gfCNCPoint6[4861] = {X 129.4526, Y 19.2665, Z -8.0000, A 0.000, B 0.000, C 0.000 }
gfCNCPoint6[4862] = {X 129.1449, Y 18.3872, Z -8.0000, A 0.000, B 0.000, C 0.000 }
gfCNCPoint6[4863] = {X 129.0406, Y 17.4615, Z -8.0000, A 0.000, B 0.000, C 0.000 }
gfCNCPoint6[4864] = {X 129.0406, Y 10.4835, Z -8.0000, A 0.000, B 0.000, C 0.000 }
gfCNCPoint6[4865] = {X 129.1435, Y 9.5642, Z -8.0000, A 0.000, B 0.000, C 0.000 }
gfCNCPoint6[4866] = {X 129.4469, Y 8.6904, Z -8.0000, A 0.000, B 0.000, C 0.000 }
gfCNCPoint6[4867] = {X 129.9360, Y 7.9052, Z -8.0000, A 0.000, B 0.000, C 0.000 }
gfCNCPoint6[4868] = {X 130.5864, Y 7.2475, Z -8.0000, A 0.000, B 0.000, C 0.000 }
gfCNCPoint6[4869] = {X 131.3662, Y 6.7499, Z -8.0000, A 0.000, B 0.000, C 0.000 }
gfCNCPoint6[4870] = {X 132.2366, Y 6.4368, Z -8.0000, A 0.000, B 0.000, C 0.000 }
gfCNCPoint6[4871] = {X 133.1547, Y 6.3238, Z -8.0000, A 0.000, B 0.000, C 0.000 }
gfCNCPoint6[4872] = {X 133.8850, Y 6.3237, Z -8.0000, A 0.000, B 0.000, C 0.000 }
gfCNCPoint6[4873] = {X 134.6950, Y 6.4118, Z -8.0000, A 0.000, B 0.000, C 0.000 }
gfCNCPoint6[4874] = {X 135.4723, Y 6.6562, Z -8.0000, A 0.000, B 0.000, C 0.000 }
gfCNCPoint6[4875] = {X 136.1871, Y 7.0473, Z -8.0000, A 0.000, B 0.000, C 0.000 }
gfCNCPoint6[4876] = {X 136.8119, Y 7.5703, Z -8.0000, A 0.000, B 0.000, C 0.000 }
gfCNCPoint6[4877] = {X 137.3228, Y 8.2050, Z -8.0000, A 0.000, B 0.000, C 0.000 }
gfCNCPoint6[4878] = {X 155.1990, Y 8.2064, Z -8.0000, A 0.000, B 0.000, C 0.000 }
gfCNCPoint6[4879] = {X 155.7105, Y 7.5705, Z -8.0000, A 0.000, B 0.000, C 0.000 }
gfCNCPoint6[4880] = {X 156.3364, Y 7.0468, Z -8.0000, A 0.000, B 0.000, C 0.000 }
gfCNCPoint6[4881] = {X 157.0525, Y 6.6553, Z -8.0000, A 0.000, B 0.000, C 0.000 }
gfCNCPoint6[4882] = {X 157.8313, Y 6.4111, Z -8.0000, A 0.000, B 0.000, C 0.000 }
gfCNCPoint6[4883] = {X 158.6427, Y 6.3237, Z -8.0000, A 0.000, B 0.000, C 0.000 }
gfCNCPoint6[4884] = {X 159.3760, Y 6.3239, Z -8.0000, A 0.000, B 0.000, C 0.000 }
gfCNCPoint6[4885] = {X 160.2928, Y 6.4383, Z -8.0000, A 0.000, B 0.000, C 0.000 }
gfCNCPoint6[4886] = {X 161.1617, Y 6.7524, Z -8.0000, A 0.000, B 0.000, C 0.000 }
gfCNCPoint6[4887] = {X 161.9398, Y 7.2504, Z -8.0000, A 0.000, B 0.000, C 0.000 }
gfCNCPoint6[4888] = {X 162.5889, Y 7.9079, Z -8.0000, A 0.000, B 0.000, C 0.000 }
gfCNCPoint6[4889] = {X 163.0768, Y 8.6925, Z -8.0000, A 0.000, B 0.000, C 0.000 }
gfCNCPoint6[4890] = {X 163.3795, Y 9.5653, Z -8.0000, A 0.000, B 0.000, C 0.000 }
gfCNCPoint6[4891] = {X 163.4821, Y 10.4835, Z -8.0000, A 0.000, B 0.000, C 0.000 }
gfCNCPoint6[4892] = {X 163.4821, Y 17.4615, Z -8.0000, A 0.000, B 0.000, C 0.000 }
gfCNCPoint6[4893] = {X 163.3795, Y 18.3798, Z -8.0000, A 0.000, B 0.000, C 0.000 }
gfCNCPoint6[4894] = {X 163.0767, Y 19.2527, Z -8.0000, A 0.000, B 0.000, C 0.000 }
gfCNCPoint6[4895] = {X 162.5887, Y 20.0373, Z -8.0000, A 0.000, B 0.000, C 0.000 }
gfCNCPoint6[4896] = {X 161.9396, Y 20.6948, Z -8.0000, A 0.000, B 0.000, C 0.000 }
gfCNCPoint6[4897] = {X 161.1613, Y 21.1929, Z -8.0000, A 0.000, B 0.000, C 0.000 }
gfCNCPoint6[4898] = {X 160.2923, Y 21.5068, Z -8.0000, A 0.000, B 0.000, C 0.000 }
gfCNCPoint6[4899] = {X 159.3755, Y 21.6212, Z -8.0000, A 0.000, B 0.000, C 0.000 }
gfCNCPoint6[4900] = {X 158.6800, Y 21.6215, Z -8.0000, A 0.000, B 0.000, C 0.000 }
gfCNCPoint6[4901] = {X 157.8559, Y 21.5370, Z -8.0000, A 0.000, B 0.000, C 0.000 }
gfCNCPoint6[4902] = {X 157.0645, Y 21.2919, Z -8.0000, A 0.000, B 0.000, C 0.000 }
gfCNCPoint6[4903] = {X 156.3369, Y 20.8959, Z -8.0000, A 0.000, B 0.000, C 0.000 }
gfCNCPoint6[4904] = {X 155.7014, Y 20.3644, Z -8.0000, A 0.000, B 0.000, C 0.000 }
gfCNCPoint6[4905] = {X 155.1830, Y 19.7182, Z -8.0000, A 0.000, B 0.000, C 0.000 }
gfCNCPoint6[4906] = {X 152.1174, Y 19.7191, Z -8.0000, A 0.000, B 0.000, C 0.000 }
gfCNCPoint6[4907] = {X 152.1164, Y 40.9370, Z -8.0000, A 0.000, B 0.000, C 0.000 }
gfCNCPoint6[4908] = {X 152.6208, Y 41.4801, Z -8.0000, A 0.000, B 0.000, C 0.000 }
gfCNCPoint6[4909] = {X 152.7136, Y 41.5904, Z -8.0000, A 0.000, B 0.000, C 0.000 }
gfCNCPoint6[4910] = {X 153.2194, Y 42.3850, Z -8.0000, A 0.000, B 0.000, C 0.000 }
gfCNCPoint6[4911] = {X 153.5346, Y 43.2727, Z -8.0000, A 0.000, B 0.000, C 0.000 }
gfCNCPoint6[4912] = {X 153.6431, Y 44.2084, Z -8.0000, A 0.000, B 0.000, C 0.000 }
gfCNCPoint6[4913] = {X 153.6429, Y 45.0400, Z -8.0000, A 0.000, B 0.000, C 0.000 }
gfCNCPoint6[4914] = {X 153.5310, Y 45.9591, Z -8.0000, A 0.000, B 0.000, C 0.000 }
gfCNCPoint6[4915] = {X 153.2186, Y 46.8306, Z -8.0000, A 0.000, B 0.000, C 0.000 }
gfCNCPoint6[4916] = {X 152.7212, Y 47.6115, Z -8.0000, A 0.000, B 0.000, C 0.000 }
gfCNCPoint6[4917] = {X 152.0634, Y 48.2631, Z -8.0000, A 0.000, B 0.000, C 0.000 }
gfCNCPoint6[4918] = {X 151.2778, Y 48.7530, Z -8.0000, A 0.000, B 0.000, C 0.000 }
gfCNCPoint6[4919] = {X 150.4032, Y 49.0570, Z -8.0000, A 0.000, B 0.000, C 0.000 }
gfCNCPoint6[4920] = {X 149.4831, Y 49.1600, Z -8.0000, A 0.000, B 0.000, C 0.000 }
gfCNCPoint6[4921] = {X 143.0396, Y 49.1600, Z -8.0000, A 0.000, B 0.000, C 0.000 }
gfCNCPoint6[4922] = {X 142.1185, Y 49.0567, Z -8.0000, A 0.000, B 0.000, C 0.000 }
gfCNCPoint6[4923] = {X 141.2432, Y 48.7521, Z -8.0000, A 0.000, B 0.000, C 0.000 }
gfCNCPoint6[4924] = {X 140.4570, Y 48.2612, Z -8.0000, A 0.000, B 0.000, C 0.000 }
gfCNCPoint6[4925] = {X 139.7990, Y 47.6084, Z -8.0000, A 0.000, B 0.000, C 0.000 }
gfCNCPoint6[4926] = {X 139.3019, Y 46.8261, Z -8.0000, A 0.000, B 0.000, C 0.000 }
gfCNCPoint6[4927] = {X 138.9903, Y 45.9532, Z -8.0000, A 0.000, B 0.000, C 0.000 }
gfCNCPoint6[4928] = {X 138.8798, Y 45.0329, Z -8.0000, A 0.000, B 0.000, C 0.000 }
gfCNCPoint6[4929] = {X 138.8800, Y 44.1516, Z -8.0000, A 0.000, B 0.000, C 0.000 }
gfCNCPoint6[4930] = {X 138.9906, Y 43.2545, Z -8.0000, A 0.000, B 0.000, C 0.000 }
gfCNCPoint6[4931] = {X 139.2922, Y 42.4026, Z -8.0000, A 0.000, B 0.000, C 0.000 }
gfCNCPoint6[4932] = {X 139.7708, Y 41.6358, Z -8.0000, A 0.000, B 0.000, C 0.000 }
gfCNCPoint6[4933] = {X 140.4036, Y 40.9906, Z -8.0000, A 0.000, B 0.000, C 0.000 }
gfCNCPoint6[4934] = {X 140.4036, Y 30.3971, Z -8.0000, A 0.000, B 0.000, C 0.000 }
gfCNCPoint6[4935] = {X 136.4036, Y 30.3971, Z -8.0000, A 0.000, B 0.000, C 0.000 }
gfCNCPoint6[4936] = {X 140.4836, Y 30.3971, Z -8.0000, A 0.000, B 0.000, C 0.000 }
gfCNCPoint6[4937] = {X 140.4836, Y 19.6385, Z -8.0000, A 0.000, B 0.000, C 0.000 }
gfCNCPoint6[4938] = {X 137.2911, Y 19.6382, Z -8.0000, A 0.000, B 0.000, C 0.000 }
gfCNCPoint6[4939] = {X 137.2218, Y 19.7475, Z -8.0000, A 0.000, B 0.000, C 0.000 }
gfCNCPoint6[4940] = {X 136.5756, Y 20.4907, Z -8.0000, A 0.000, B 0.000, C 0.000 }
gfCNCPoint6[4941] = {X 135.7702, Y 21.0573, Z -8.0000, A 0.000, B 0.000, C 0.000 }
gfCNCPoint6[4942] = {X 134.8524, Y 21.4145, Z -8.0000, A 0.000, B 0.000, C 0.000 }
gfCNCPoint6[4943] = {X 133.8758, Y 21.5414, Z -8.0000, A 0.000, B 0.000, C 0.000 }
gfCNCPoint6[4944] = {X 133.2006, Y 21.5415, Z -8.0000, A 0.000, B 0.000, C 0.000 }
gfCNCPoint6[4945] = {X 132.2928, Y 21.4392, Z -8.0000, A 0.000, B 0.000, C 0.000 }
gfCNCPoint6[4946] = {X 131.4304, Y 21.1375, Z -8.0000, A 0.000, B 0.000, C 0.000 }
gfCNCPoint6[4947] = {X 130.6568, Y 20.6514, Z -8.0000, A 0.000, B 0.000, C 0.000 }
gfCNCPoint6[4948] = {X 130.0108, Y 20.0054, Z -8.0000, A 0.000, B 0.000, C 0.000 }
gfCNCPoint6[4949] = {X 129.5247, Y 19.2318, Z -8.0000, A 0.000, B 0.000, C 0.000 }
gfCNCPoint6[4950] = {X 129.2229, Y 18.3694, Z -8.0000, A 0.000, B 0.000, C 0.000 }
gfCNCPoint6[4951] = {X 129.1206, Y 17.4615, Z -8.0000, A 0.000, B 0.000, C 0.000 }
gfCNCPoint6[4952] = {X 129.1206, Y 10.4835, Z -8.0000, A 0.000, B 0.000, C 0.000 }
gfCNCPoint6[4953] = {X 129.2215, Y 9.5820, Z -8.0000, A 0.000, B 0.000, C 0.000 }
gfCNCPoint6[4954] = {X 129.5191, Y 8.7250, Z -8.0000, A 0.000, B 0.000, C 0.000 }
gfCNCPoint6[4955] = {X 129.9986, Y 7.9550, Z -8.0000, A 0.000, B 0.000, C 0.000 }
gfCNCPoint6[4956] = {X 130.6365, Y 7.3099, Z -8.0000, A 0.000, B 0.000, C 0.000 }
gfCNCPoint6[4957] = {X 131.4011, Y 6.8218, Z -8.0000, A 0.000, B 0.000, C 0.000 }
gfCNCPoint6[4958] = {X 132.2547, Y 6.5147, Z -8.0000, A 0.000, B 0.000, C 0.000 }
gfCNCPoint6[4959] = {X 133.1551, Y 6.4038, Z -8.0000, A 0.000, B 0.000, C 0.000 }
gfCNCPoint6[4960] = {X 133.8841, Y 6.4037, Z -8.0000, A 0.000, B 0.000, C 0.000 }
gfCNCPoint6[4961] = {X 134.6870, Y 6.4919, Z -8.0000, A 0.000, B 0.000, C 0.000 }
gfCNCPoint6[4962] = {X 135.4568, Y 6.7365, Z -8.0000, A 0.000, B 0.000, C 0.000 }
gfCNCPoint6[4963] = {X 136.1633, Y 7.1280, Z -8.0000, A 0.000, B 0.000, C 0.000 }
gfCNCPoint6[4964] = {X 136.7789, Y 7.6510, Z -8.0000, A 0.000, B 0.000, C 0.000 }
gfCNCPoint6[4965] = {X 137.2793, Y 8.2850, Z -8.0000, A 0.000, B 0.000, C 0.000 }
gfCNCPoint6[4966] = {X 155.2425, Y 8.2864, Z -8.0000, A 0.000, B 0.000, C 0.000 }
gfCNCPoint6[4967] = {X 155.2880, Y 8.2168, Z -8.0000, A 0.000, B 0.000, C 0.000 }
gfCNCPoint6[4968] = {X 155.3349, Y 8.1482, Z -8.0000, A 0.000, B 0.000, C 0.000 }
gfCNCPoint6[4969] = {X 155.9800, Y 7.4251, Z -8.0000, A 0.000, B 0.000, C 0.000 }
gfCNCPoint6[4970] = {X 156.7775, Y 6.8745, Z -8.0000, A 0.000, B 0.000, C 0.000 }
gfCNCPoint6[4971] = {X 157.6823, Y 6.5275, Z -8.0000, A 0.000, B 0.000, C 0.000 }
gfCNCPoint6[4972] = {X 158.6434, Y 6.4037, Z -8.0000, A 0.000, B 0.000, C 0.000 }
gfCNCPoint6[4973] = {X 159.3750, Y 6.4039, Z -8.0000, A 0.000, B 0.000, C 0.000 }
gfCNCPoint6[4974] = {X 160.2741, Y 6.5161, Z -8.0000, A 0.000, B 0.000, C 0.000 }
gfCNCPoint6[4975] = {X 161.1263, Y 6.8241, Z -8.0000, A 0.000, B 0.000, C 0.000 }
gfCNCPoint6[4976] = {X 161.8895, Y 7.3126, Z -8.0000, A 0.000, B 0.000, C 0.000 }
gfCNCPoint6[4977] = {X 162.5260, Y 7.9574, Z -8.0000, A 0.000, B 0.000, C 0.000 }
gfCNCPoint6[4978] = {X 163.0046, Y 8.7269, Z -8.0000, A 0.000, B 0.000, C 0.000 }
gfCNCPoint6[4979] = {X 163.3015, Y 9.5830, Z -8.0000, A 0.000, B 0.000, C 0.000 }
gfCNCPoint6[4980] = {X 163.4021, Y 10.4835, Z -8.0000, A 0.000, B 0.000, C 0.000 }
gfCNCPoint6[4981] = {X 163.4021, Y 17.4615, Z -8.0000, A 0.000, B 0.000, C 0.000 }
gfCNCPoint6[4982] = {X 163.3015, Y 18.3621, Z -8.0000, A 0.000, B 0.000, C 0.000 }
gfCNCPoint6[4983] = {X 163.0046, Y 19.2182, Z -8.0000, A 0.000, B 0.000, C 0.000 }
gfCNCPoint6[4984] = {X 162.5260, Y 19.9876, Z -8.0000, A 0.000, B 0.000, C 0.000 }
gfCNCPoint6[4985] = {X 161.8895, Y 20.6325, Z -8.0000, A 0.000, B 0.000, C 0.000 }
gfCNCPoint6[4986] = {X 161.1263, Y 21.1209, Z -8.0000, A 0.000, B 0.000, C 0.000 }
gfCNCPoint6[4987] = {X 160.2741, Y 21.4289, Z -8.0000, A 0.000, B 0.000, C 0.000 }
gfCNCPoint6[4988] = {X 159.3750, Y 21.5412, Z -8.0000, A 0.000, B 0.000, C 0.000 }
gfCNCPoint6[4989] = {X 158.6802, Y 21.5415, Z -8.0000, A 0.000, B 0.000, C 0.000 }
gfCNCPoint6[4990] = {X 157.8634, Y 21.4569, Z -8.0000, A 0.000, B 0.000, C 0.000 }
gfCNCPoint6[4991] = {X 157.0797, Y 21.2114, Z -8.0000, A 0.000, B 0.000, C 0.000 }
gfCNCPoint6[4992] = {X 156.3605, Y 20.8151, Z -8.0000, A 0.000, B 0.000, C 0.000 }
gfCNCPoint6[4993] = {X 155.7345, Y 20.2836, Z -8.0000, A 0.000, B 0.000, C 0.000 }
gfCNCPoint6[4994] = {X 155.2267, Y 19.6382, Z -8.0000, A 0.000, B 0.000, C 0.000 }
gfCNCPoint6[4995] = {X 152.0374, Y 19.6392, Z -8.0000, A 0.000, B 0.000, C 0.000 }
gfCNCPoint6[4996] = {X 152.0364, Y 40.9685, Z -8.0000, A 0.000, B 0.000, C 0.000 }
gfCNCPoint6[4997] = {X 152.5609, Y 41.5331, Z -8.0000, A 0.000, B 0.000, C 0.000 }
gfCNCPoint6[4998] = {X 152.6518, Y 41.6413, Z -8.0000, A 0.000, B 0.000, C 0.000 }
gfCNCPoint6[4999] = {X 153.1477, Y 42.4206, Z -8.0000, A 0.000, B 0.000, C 0.000 }
gfCNCPoint6[5000] = {X 153.4567, Y 43.2911, Z -8.0000, A 0.000, B 0.000, C 0.000 }
gfCNCPoint6[5001] = {X 153.5631, Y 44.2086, Z -8.0000, A 0.000, B 0.000, C 0.000 }
gfCNCPoint6[5002] = {X 153.5629, Y 45.0392, Z -8.0000, A 0.000, B 0.000, C 0.000 }
gfCNCPoint6[5003] = {X 153.4532, Y 45.9406, Z -8.0000, A 0.000, B 0.000, C 0.000 }
gfCNCPoint6[5004] = {X 153.1468, Y 46.7954, Z -8.0000, A 0.000, B 0.000, C 0.000 }
gfCNCPoint6[5005] = {X 152.6589, Y 47.5613, Z -8.0000, A 0.000, B 0.000, C 0.000 }
gfCNCPoint6[5006] = {X 152.0138, Y 48.2003, Z -8.0000, A 0.000, B 0.000, C 0.000 }
gfCNCPoint6[5007] = {X 151.2432, Y 48.6808, Z -8.0000, A 0.000, B 0.000, C 0.000 }
gfCNCPoint6[5008] = {X 150.3855, Y 48.9789, Z -8.0000, A 0.000, B 0.000, C 0.000 }
gfCNCPoint6[5009] = {X 149.4831, Y 49.0800, Z -8.0000, A 0.000, B 0.000, C 0.000 }
gfCNCPoint6[5010] = {X 143.0396, Y 49.0800, Z -8.0000, A 0.000, B 0.000, C 0.000 }
gfCNCPoint6[5011] = {X 142.1362, Y 48.9787, Z -8.0000, A 0.000, B 0.000, C 0.000 }
gfCNCPoint6[5012] = {X 141.2777, Y 48.6799, Z -8.0000, A 0.000, B 0.000, C 0.000 }
gfCNCPoint6[5013] = {X 140.5066, Y 48.1985, Z -8.0000, A 0.000, B 0.000, C 0.000 }
gfCNCPoint6[5014] = {X 139.8613, Y 47.5582, Z -8.0000, A 0.000, B 0.000, C 0.000 }
gfCNCPoint6[5015] = {X 139.3737, Y 46.7910, Z -8.0000, A 0.000, B 0.000, C 0.000 }
gfCNCPoint6[5016] = {X 139.0682, Y 45.9349, Z -8.0000, A 0.000, B 0.000, C 0.000 }
gfCNCPoint6[5017] = {X 138.9598, Y 45.0323, Z -8.0000, A 0.000, B 0.000, C 0.000 }
gfCNCPoint6[5018] = {X 138.9600, Y 44.1527, Z -8.0000, A 0.000, B 0.000, C 0.000 }
gfCNCPoint6[5019] = {X 139.0706, Y 43.2637, Z -8.0000, A 0.000, B 0.000, C 0.000 }
gfCNCPoint6[5020] = {X 139.3725, Y 42.4203, Z -8.0000, A 0.000, B 0.000, C 0.000 }
gfCNCPoint6[5021] = {X 139.8512, Y 41.6631, Z -8.0000, A 0.000, B 0.000, C 0.000 }
gfCNCPoint6[5022] = {X 140.4836, Y 41.0287, Z -8.0000, A 0.000, B 0.000, C 0.000 }
gfCNCPoint6[5023] = {X 140.4836, Y 30.3971, Z -8.0000, A 0.000, B 0.000, C 0.000 }
gfCNCPoint6[5024] = {X 136.4836, Y 30.3971, Z -8.0000, A 0.000, B 0.000, C 0.000 }
gfCNCPoint6[5025] = {X 140.5636, Y 30.3971, Z -8.0000, A 0.000, B 0.000, C 0.000 }
gfCNCPoint6[5026] = {X 140.5636, Y 19.5585, Z -8.0000, A 0.000, B 0.000, C 0.000 }
gfCNCPoint6[5027] = {X 137.2663, Y 19.5582, Z -8.0000, A 0.000, B 0.000, C 0.000 }
gfCNCPoint6[5028] = {X 137.2447, Y 19.5621, Z -8.0000, A 0.000, B 0.000, C 0.000 }
gfCNCPoint6[5029] = {X 137.1360, Y 19.7312, Z -8.0000, A 0.000, B 0.000, C 0.000 }
gfCNCPoint6[5030] = {X 136.4965, Y 20.4541, Z -8.0000, A 0.000, B 0.000, C 0.000 }
gfCNCPoint6[5031] = {X 135.7025, Y 21.0027, Z -8.0000, A 0.000, B 0.000, C 0.000 }
gfCNCPoint6[5032] = {X 134.8003, Y 21.3451, Z -8.0000, A 0.000, B 0.000, C 0.000 }
gfCNCPoint6[5033] = {X 133.8422, Y 21.4615, Z -8.0000, A 0.000, B 0.000, C 0.000 }
gfCNCPoint6[5034] = {X 133.2006, Y 21.4615, Z -8.0000, A 0.000, B 0.000, C 0.000 }
gfCNCPoint6[5035] = {X 132.3106, Y 21.3612, Z -8.0000, A 0.000, B 0.000, C 0.000 }
gfCNCPoint6[5036] = {X 131.4651, Y 21.0654, Z -8.0000, A 0.000, B 0.000, C 0.000 }
gfCNCPoint6[5037] = {X 130.7067, Y 20.5889, Z -8.0000, A 0.000, B 0.000, C 0.000 }
gfCNCPoint6[5038] = {X 130.0733, Y 19.9555, Z -8.0000, A 0.000, B 0.000, C 0.000 }
gfCNCPoint6[5039] = {X 129.5968, Y 19.1971, Z -8.0000, A 0.000, B 0.000, C 0.000 }
gfCNCPoint6[5040] = {X 129.3009, Y 18.3516, Z -8.0000, A 0.000, B 0.000, C 0.000 }
gfCNCPoint6[5041] = {X 129.2006, Y 17.4615, Z -8.0000, A 0.000, B 0.000, C 0.000 }
gfCNCPoint6[5042] = {X 129.2006, Y 10.4835, Z -8.0000, A 0.000, B 0.000, C 0.000 }
gfCNCPoint6[5043] = {X 129.3009, Y 9.5934, Z -8.0000, A 0.000, B 0.000, C 0.000 }
gfCNCPoint6[5044] = {X 129.5968, Y 8.7480, Z -8.0000, A 0.000, B 0.000, C 0.000 }
gfCNCPoint6[5045] = {X 130.0733, Y 7.9896, Z -8.0000, A 0.000, B 0.000, C 0.000 }
gfCNCPoint6[5046] = {X 130.7067, Y 7.3562, Z -8.0000, A 0.000, B 0.000, C 0.000 }
gfCNCPoint6[5047] = {X 131.4651, Y 6.8796, Z -8.0000, A 0.000, B 0.000, C 0.000 }
gfCNCPoint6[5048] = {X 132.3106, Y 6.5838, Z -8.0000, A 0.000, B 0.000, C 0.000 }
gfCNCPoint6[5049] = {X 133.2007, Y 6.4835, Z -8.0000, A 0.000, B 0.000, C 0.000 }
gfCNCPoint6[5050] = {X 133.8833, Y 6.4837, Z -8.0000, A 0.000, B 0.000, C 0.000 }
gfCNCPoint6[5051] = {X 134.6790, Y 6.5720, Z -8.0000, A 0.000, B 0.000, C 0.000 }
gfCNCPoint6[5052] = {X 135.4412, Y 6.8170, Z -8.0000, A 0.000, B 0.000, C 0.000 }
gfCNCPoint6[5053] = {X 136.1393, Y 7.2088, Z -8.0000, A 0.000, B 0.000, C 0.000 }
gfCNCPoint6[5054] = {X 136.7454, Y 7.7318, Z -8.0000, A 0.000, B 0.000, C 0.000 }
gfCNCPoint6[5055] = {X 137.2352, Y 8.3650, Z -8.0000, A 0.000, B 0.000, C 0.000 }
gfCNCPoint6[5056] = {X 155.2276, Y 8.3650, Z -8.0000, A 0.000, B 0.000, C 0.000 }
gfCNCPoint6[5057] = {X 155.2814, Y 8.3748, Z -8.0000, A 0.000, B 0.000, C 0.000 }
gfCNCPoint6[5058] = {X 155.3397, Y 8.2836, Z -8.0000, A 0.000, B 0.000, C 0.000 }
gfCNCPoint6[5059] = {X 155.4005, Y 8.1940, Z -8.0000, A 0.000, B 0.000, C 0.000 }
gfCNCPoint6[5060] = {X 156.0398, Y 7.4790, Z -8.0000, A 0.000, B 0.000, C 0.000 }
gfCNCPoint6[5061] = {X 156.8309, Y 6.9368, Z -8.0000, A 0.000, B 0.000, C 0.000 }
gfCNCPoint6[5062] = {X 157.7283, Y 6.5985, Z -8.0000, A 0.000, B 0.000, C 0.000 }
gfCNCPoint6[5063] = {X 158.6805, Y 6.4835, Z -8.0000, A 0.000, B 0.000, C 0.000 }
gfCNCPoint6[5064] = {X 159.3739, Y 6.4839, Z -8.0000, A 0.000, B 0.000, C 0.000 }
gfCNCPoint6[5065] = {X 160.2554, Y 6.5939, Z -8.0000, A 0.000, B 0.000, C 0.000 }
gfCNCPoint6[5066] = {X 161.0909, Y 6.8959, Z -8.0000, A 0.000, B 0.000, C 0.000 }
gfCNCPoint6[5067] = {X 161.8391, Y 7.3747, Z -8.0000, A 0.000, B 0.000, C 0.000 }
gfCNCPoint6[5068] = {X 162.4632, Y 8.0070, Z -8.0000, A 0.000, B 0.000, C 0.000 }
gfCNCPoint6[5069] = {X 162.9324, Y 8.7613, Z -8.0000, A 0.000, B 0.000, C 0.000 }
gfCNCPoint6[5070] = {X 163.2234, Y 9.6007, Z -8.0000, A 0.000, B 0.000, C 0.000 }
gfCNCPoint6[5071] = {X 163.3221, Y 10.4835, Z -8.0000, A 0.000, B 0.000, C 0.000 }
gfCNCPoint6[5072] = {X 163.3221, Y 17.4615, Z -8.0000, A 0.000, B 0.000, C 0.000 }
gfCNCPoint6[5073] = {X 163.2218, Y 18.3516, Z -8.0000, A 0.000, B 0.000, C 0.000 }
gfCNCPoint6[5074] = {X 162.9260, Y 19.1971, Z -8.0000, A 0.000, B 0.000, C 0.000 }
gfCNCPoint6[5075] = {X 162.4494, Y 19.9555, Z -8.0000, A 0.000, B 0.000, C 0.000 }
gfCNCPoint6[5076] = {X 161.8160, Y 20.5889, Z -8.0000, A 0.000, B 0.000, C 0.000 }
gfCNCPoint6[5077] = {X 161.0576, Y 21.0654, Z -8.0000, A 0.000, B 0.000, C 0.000 }
gfCNCPoint6[5078] = {X 160.2122, Y 21.3613, Z -8.0000, A 0.000, B 0.000, C 0.000 }
gfCNCPoint6[5079] = {X 159.3221, Y 21.4615, Z -8.0000, A 0.000, B 0.000, C 0.000 }
gfCNCPoint6[5080] = {X 158.6805, Y 21.4615, Z -8.0000, A 0.000, B 0.000, C 0.000 }
gfCNCPoint6[5081] = {X 157.8710, Y 21.3767, Z -8.0000, A 0.000, B 0.000, C 0.000 }
gfCNCPoint6[5082] = {X 157.0950, Y 21.1310, Z -8.0000, A 0.000, B 0.000, C 0.000 }
gfCNCPoint6[5083] = {X 156.3843, Y 20.7342, Z -8.0000, A 0.000, B 0.000, C 0.000 }
gfCNCPoint6[5084] = {X 155.7679, Y 20.2027, Z -8.0000, A 0.000, B 0.000, C 0.000 }
gfCNCPoint6[5085] = {X 155.2709, Y 19.5582, Z -8.0000, A 0.000, B 0.000, C 0.000 }
gfCNCPoint6[5086] = {X 151.9574, Y 19.5592, Z -8.0000, A 0.000, B 0.000, C 0.000 }
gfCNCPoint6[5087] = {X 151.9564, Y 40.9999, Z -8.0000, A 0.000, B 0.000, C 0.000 }
gfCNCPoint6[5088] = {X 152.5009, Y 41.5861, Z -8.0000, A 0.000, B 0.000, C 0.000 }
gfCNCPoint6[5089] = {X 152.5901, Y 41.6922, Z -8.0000, A 0.000, B 0.000, C 0.000 }
gfCNCPoint6[5090] = {X 153.0761, Y 42.4561, Z -8.0000, A 0.000, B 0.000, C 0.000 }
gfCNCPoint6[5091] = {X 153.3788, Y 43.3094, Z -8.0000, A 0.000, B 0.000, C 0.000 }
gfCNCPoint6[5092] = {X 153.4831, Y 44.2088, Z -8.0000, A 0.000, B 0.000, C 0.000 }
gfCNCPoint6[5093] = {X 153.4829, Y 45.0384, Z -8.0000, A 0.000, B 0.000, C 0.000 }
gfCNCPoint6[5094] = {X 153.3753, Y 45.9222, Z -8.0000, A 0.000, B 0.000, C 0.000 }
gfCNCPoint6[5095] = {X 153.0750, Y 46.7602, Z -8.0000, A 0.000, B 0.000, C 0.000 }
gfCNCPoint6[5096] = {X 152.5967, Y 47.5111, Z -8.0000, A 0.000, B 0.000, C 0.000 }
gfCNCPoint6[5097] = {X 151.9642, Y 48.1376, Z -8.0000, A 0.000, B 0.000, C 0.000 }
gfCNCPoint6[5098] = {X 151.2087, Y 48.6086, Z -8.0000, A 0.000, B 0.000, C 0.000 }
gfCNCPoint6[5099] = {X 150.3678, Y 48.9009, Z -8.0000, A 0.000, B 0.000, C 0.000 }
gfCNCPoint6[5100] = {X 149.4831, Y 49.0000, Z -8.0000, A 0.000, B 0.000, C 0.000 }
gfCNCPoint6[5101] = {X 143.0396, Y 49.0000, Z -8.0000, A 0.000, B 0.000, C 0.000 }
gfCNCPoint6[5102] = {X 142.1495, Y 48.8997, Z -8.0000, A 0.000, B 0.000, C 0.000 }
gfCNCPoint6[5103] = {X 141.3041, Y 48.6039, Z -8.0000, A 0.000, B 0.000, C 0.000 }
gfCNCPoint6[5104] = {X 140.5457, Y 48.1273, Z -8.0000, A 0.000, B 0.000, C 0.000 }
gfCNCPoint6[5105] = {X 139.9123, Y 47.4939, Z -8.0000, A 0.000, B 0.000, C 0.000 }
gfCNCPoint6[5106] = {X 139.4357, Y 46.7355, Z -8.0000, A 0.000, B 0.000, C 0.000 }
gfCNCPoint6[5107] = {X 139.1399, Y 45.8901, Z -8.0000, A 0.000, B 0.000, C 0.000 }
gfCNCPoint6[5108] = {X 139.0396, Y 45.0000, Z -8.0000, A 0.000, B 0.000, C 0.000 }
gfCNCPoint6[5109] = {X 139.0400, Y 44.1538, Z -8.0000, A 0.000, B 0.000, C 0.000 }
gfCNCPoint6[5110] = {X 139.1506, Y 43.2730, Z -8.0000, A 0.000, B 0.000, C 0.000 }
gfCNCPoint6[5111] = {X 139.4528, Y 42.4382, Z -8.0000, A 0.000, B 0.000, C 0.000 }
gfCNCPoint6[5112] = {X 139.9317, Y 41.6907, Z -8.0000, A 0.000, B 0.000, C 0.000 }
gfCNCPoint6[5113] = {X 140.5636, Y 41.0672, Z -8.0000, A 0.000, B 0.000, C 0.000 }
gfCNCPoint6[5114] = {X 140.5636, Y 30.3971, Z -8.0000, A 0.000, B 0.000, C 0.000 }
gfCNCPoint6[5115] = {X 136.4836, Y 30.3971, Z -8.0000, A 0.000, B 0.000, C 0.000 }
gfCNCPoint6[5116] = {X 136.4836, Y 30.3971, Z -5.0000, A 0.000, B 0.000, C 0.000 }
gfCNCPoint6[5117] = {X 136.4836, Y 30.3971, Z 11.0000, A 0.000, B 0.000, C 0.000 }
gfCNCPoint6[5118] = {X 137.6628, Y 74.8910, Z 11.0000, A 0.000, B 0.000, C 0.000 }
gfCNCPoint6[5119] = {X 137.6628, Y 74.8910, Z -5.0000, A 0.000, B 0.000, C 0.000 }
gfCNCPoint6[5120] = {X 137.6628, Y 74.8910, Z -8.0000, A 0.000, B 0.000, C 0.000 }
gfCNCPoint6[5121] = {X 140.6793, Y 77.6382, Z -8.0000, A 0.000, B 0.000, C 0.000 }
gfCNCPoint6[5122] = {X 155.6319, Y 61.2193, Z -8.0000, A 0.000, B 0.000, C 0.000 }
gfCNCPoint6[5123] = {X 155.2772, Y 60.5138, Z -8.0000, A 0.000, B 0.000, C 0.000 }
gfCNCPoint6[5124] = {X 155.0568, Y 59.7555, Z -8.0000, A 0.000, B 0.000, C 0.000 }
gfCNCPoint6[5125] = {X 154.9781, Y 58.9697, Z -8.0000, A 0.000, B 0.000, C 0.000 }
gfCNCPoint6[5126] = {X 154.9780, Y 58.0000, Z -8.0000, A 0.000, B 0.000, C 0.000 }
gfCNCPoint6[5127] = {X 155.0863, Y 57.0387, Z -8.0000, A 0.000, B 0.000, C 0.000 }
gfCNCPoint6[5128] = {X 155.4058, Y 56.1256, Z -8.0000, A 0.000, B 0.000, C 0.000 }
gfCNCPoint6[5129] = {X 155.9204, Y 55.3065, Z -8.0000, A 0.000, B 0.000, C 0.000 }
gfCNCPoint6[5130] = {X 156.6045, Y 54.6225, Z -8.0000, A 0.000, B 0.000, C 0.000 }
gfCNCPoint6[5131] = {X 157.4236, Y 54.1078, Z -8.0000, A 0.000, B 0.000, C 0.000 }
gfCNCPoint6[5132] = {X 158.3367, Y 53.7883, Z -8.0000, A 0.000, B 0.000, C 0.000 }
gfCNCPoint6[5133] = {X 159.2980, Y 53.6800, Z -8.0000, A 0.000, B 0.000, C 0.000 }
gfCNCPoint6[5134] = {X 178.5335, Y 53.6800, Z -8.0000, A 0.000, B 0.000, C 0.000 }
gfCNCPoint6[5135] = {X 179.4948, Y 53.7883, Z -8.0000, A 0.000, B 0.000, C 0.000 }
gfCNCPoint6[5136] = {X 180.4079, Y 54.1078, Z -8.0000, A 0.000, B 0.000, C 0.000 }
gfCNCPoint6[5137] = {X 181.2270, Y 54.6225, Z -8.0000, A 0.000, B 0.000, C 0.000 }
gfCNCPoint6[5138] = {X 181.9110, Y 55.3065, Z -8.0000, A 0.000, B 0.000, C 0.000 }
gfCNCPoint6[5139] = {X 182.4257, Y 56.1256, Z -8.0000, A 0.000, B 0.000, C 0.000 }
gfCNCPoint6[5140] = {X 182.7452, Y 57.0387, Z -8.0000, A 0.000, B 0.000, C 0.000 }
gfCNCPoint6[5141] = {X 182.8535, Y 58.0000, Z -8.0000, A 0.000, B 0.000, C 0.000 }
gfCNCPoint6[5142] = {X 182.8535, Y 58.9342, Z -8.0000, A 0.000, B 0.000, C 0.000 }
gfCNCPoint6[5143] = {X 182.7809, Y 59.7229, Z -8.0000, A 0.000, B 0.000, C 0.000 }
gfCNCPoint6[5144] = {X 182.5654, Y 60.4851, Z -8.0000, A 0.000, B 0.000, C 0.000 }
gfCNCPoint6[5145] = {X 182.2145, Y 61.1952, Z -8.0000, A 0.000, B 0.000, C 0.000 }
gfCNCPoint6[5146] = {X 209.2942, Y 90.7568, Z -8.0000, A 0.000, B 0.000, C 0.000 }
gfCNCPoint6[5147] = {X 209.9660, Y 91.4528, Z -8.0000, A 0.000, B 0.000, C 0.000 }
gfCNCPoint6[5148] = {X 210.6734, Y 92.1126, Z -8.0000, A 0.000, B 0.000, C 0.000 }
gfCNCPoint6[5149] = {X 211.0689, Y 92.3802, Z -8.0000, A 0.000, B 0.000, C 0.000 }
gfCNCPoint6[5150] = {X 211.5197, Y 92.5376, Z -8.0000, A 0.000, B 0.000, C 0.000 }
gfCNCPoint6[5151] = {X 212.1074, Y 92.6607, Z -8.0000, A 0.000, B 0.000, C 0.000 }
gfCNCPoint6[5152] = {X 213.3763, Y 92.8205, Z -8.0000, A 0.000, B 0.000, C 0.000 }
gfCNCPoint6[5153] = {X 214.4407, Y 92.7359, Z -8.0000, A 0.000, B 0.000, C 0.000 }
gfCNCPoint6[5154] = {X 215.5068, Y 92.6742, Z -8.0000, A 0.000, B 0.000, C 0.000 }
gfCNCPoint6[5155] = {X 216.1771, Y 92.6014, Z -8.0000, A 0.000, B 0.000, C 0.000 }
gfCNCPoint6[5156] = {X 216.8224, Y 92.4063, Z -8.0000, A 0.000, B 0.000, C 0.000 }
gfCNCPoint6[5157] = {X 217.4209, Y 92.0958, Z -8.0000, A 0.000, B 0.000, C 0.000 }
gfCNCPoint6[5158] = {X 222.9613, Y 88.5203, Z -8.0000, A 0.000, B 0.000, C 0.000 }
gfCNCPoint6[5159] = {X 245.8267, Y 73.8997, Z -8.0000, A 0.000, B 0.000, C 0.000 }
gfCNCPoint6[5160] = {X 221.6306, Y 64.4051, Z -8.0000, A 0.000, B 0.000, C 0.000 }
gfCNCPoint6[5161] = {X 219.8631, Y 63.8136, Z -8.0000, A 0.000, B 0.000, C 0.000 }
gfCNCPoint6[5162] = {X 218.0397, Y 63.4275, Z -8.0000, A 0.000, B 0.000, C 0.000 }
gfCNCPoint6[5163] = {X 216.1841, Y 63.2516, Z -8.0000, A 0.000, B 0.000, C 0.000 }
gfCNCPoint6[5164] = {X 215.2523, Y 63.1173, Z -8.0000, A 0.000, B 0.000, C 0.000 }
gfCNCPoint6[5165] = {X 214.3717, Y 62.7843, Z -8.0000, A 0.000, B 0.000, C 0.000 }
gfCNCPoint6[5166] = {X 213.5841, Y 62.2684, Z -8.0000, A 0.000, B 0.000, C 0.000 }
gfCNCPoint6[5167] = {X 212.9270, Y 61.5942, Z -8.0000, A 0.000, B 0.000, C 0.000 }
gfCNCPoint6[5168] = {X 212.4315, Y 60.7936, Z -8.0000, A 0.000, B 0.000, C 0.000 }
gfCNCPoint6[5169] = {X 212.1213, Y 59.9047, Z -8.0000, A 0.000, B 0.000, C 0.000 }
gfCNCPoint6[5170] = {X 212.0110, Y 58.9697, Z -8.0000, A 0.000, B 0.000, C 0.000 }
gfCNCPoint6[5171] = {X 212.0108, Y 58.0000, Z -8.0000, A 0.000, B 0.000, C 0.000 }
gfCNCPoint6[5172] = {X 212.1191, Y 57.0387, Z -8.0000, A 0.000, B 0.000, C 0.000 }
gfCNCPoint6[5173] = {X 212.4386, Y 56.1256, Z -8.0000, A 0.000, B 0.000, C 0.000 }
gfCNCPoint6[5174] = {X 212.9533, Y 55.3065, Z -8.0000, A 0.000, B 0.000, C 0.000 }
gfCNCPoint6[5175] = {X 213.6373, Y 54.6225, Z -8.0000, A 0.000, B 0.000, C 0.000 }
gfCNCPoint6[5176] = {X 214.4564, Y 54.1078, Z -8.0000, A 0.000, B 0.000, C 0.000 }
gfCNCPoint6[5177] = {X 215.3695, Y 53.7883, Z -8.0000, A 0.000, B 0.000, C 0.000 }
gfCNCPoint6[5178] = {X 216.3308, Y 53.6800, Z -8.0000, A 0.000, B 0.000, C 0.000 }
gfCNCPoint6[5179] = {X 237.2617, Y 53.6800, Z -8.0000, A 0.000, B 0.000, C 0.000 }
gfCNCPoint6[5180] = {X 238.2230, Y 53.7883, Z -8.0000, A 0.000, B 0.000, C 0.000 }
gfCNCPoint6[5181] = {X 239.1361, Y 54.1078, Z -8.0000, A 0.000, B 0.000, C 0.000 }
gfCNCPoint6[5182] = {X 239.9552, Y 54.6225, Z -8.0000, A 0.000, B 0.000, C 0.000 }
gfCNCPoint6[5183] = {X 240.6392, Y 55.3065, Z -8.0000, A 0.000, B 0.000, C 0.000 }
gfCNCPoint6[5184] = {X 241.1539, Y 56.1256, Z -8.0000, A 0.000, B 0.000, C 0.000 }
gfCNCPoint6[5185] = {X 241.4734, Y 57.0387, Z -8.0000, A 0.000, B 0.000, C 0.000 }
gfCNCPoint6[5186] = {X 241.5817, Y 58.0000, Z -8.0000, A 0.000, B 0.000, C 0.000 }
gfCNCPoint6[5187] = {X 241.5817, Y 58.2316, Z -8.0000, A 0.000, B 0.000, C 0.000 }
gfCNCPoint6[5188] = {X 248.1152, Y 60.7793, Z -8.0000, A 0.000, B 0.000, C 0.000 }
gfCNCPoint6[5189] = {X 275.6316, Y 71.7011, Z -8.0000, A 0.000, B 0.000, C 0.000 }
gfCNCPoint6[5190] = {X 275.6333, Y 63.2123, Z -8.0000, A 0.000, B 0.000, C 0.000 }
gfCNCPoint6[5191] = {X 274.7817, Y 63.0031, Z -8.0000, A 0.000, B 0.000, C 0.000 }
gfCNCPoint6[5192] = {X 273.9899, Y 62.6263, Z -8.0000, A 0.000, B 0.000, C 0.000 }
gfCNCPoint6[5193] = {X 273.2905, Y 62.0973, Z -8.0000, A 0.000, B 0.000, C 0.000 }
gfCNCPoint6[5194] = {X 272.7124, Y 61.4380, Z -8.0000, A 0.000, B 0.000, C 0.000 }
gfCNCPoint6[5195] = {X 272.2793, Y 60.6756, Z -8.0000, A 0.000, B 0.000, C 0.000 }
gfCNCPoint6[5196] = {X 272.0090, Y 59.8413, Z -8.0000, A 0.000, B 0.000, C 0.000 }
gfCNCPoint6[5197] = {X 271.9128, Y 58.9697, Z -8.0000, A 0.000, B 0.000, C 0.000 }
gfCNCPoint6[5198] = {X 271.9127, Y 58.0000, Z -8.0000, A 0.000, B 0.000, C 0.000 }
gfCNCPoint6[5199] = {X 272.0210, Y 57.0387, Z -8.0000, A 0.000, B 0.000, C 0.000 }
gfCNCPoint6[5200] = {X 272.3405, Y 56.1256, Z -8.0000, A 0.000, B 0.000, C 0.000 }
gfCNCPoint6[5201] = {X 272.8552, Y 55.3065, Z -8.0000, A 0.000, B 0.000, C 0.000 }
gfCNCPoint6[5202] = {X 273.5392, Y 54.6225, Z -8.0000, A 0.000, B 0.000, C 0.000 }
gfCNCPoint6[5203] = {X 274.3583, Y 54.1078, Z -8.0000, A 0.000, B 0.000, C 0.000 }
gfCNCPoint6[5204] = {X 275.2714, Y 53.7883, Z -8.0000, A 0.000, B 0.000, C 0.000 }
gfCNCPoint6[5205] = {X 276.2327, Y 53.6800, Z -8.0000, A 0.000, B 0.000, C 0.000 }
gfCNCPoint6[5206] = {X 292.7731, Y 53.6800, Z -8.0000, A 0.000, B 0.000, C 0.000 }
gfCNCPoint6[5207] = {X 293.7344, Y 53.7883, Z -8.0000, A 0.000, B 0.000, C 0.000 }
gfCNCPoint6[5208] = {X 294.6475, Y 54.1078, Z -8.0000, A 0.000, B 0.000, C 0.000 }
gfCNCPoint6[5209] = {X 295.4666, Y 54.6225, Z -8.0000, A 0.000, B 0.000, C 0.000 }
gfCNCPoint6[5210] = {X 296.1506, Y 55.3065, Z -8.0000, A 0.000, B 0.000, C 0.000 }
gfCNCPoint6[5211] = {X 296.6653, Y 56.1256, Z -8.0000, A 0.000, B 0.000, C 0.000 }
gfCNCPoint6[5212] = {X 296.9848, Y 57.0387, Z -8.0000, A 0.000, B 0.000, C 0.000 }
gfCNCPoint6[5213] = {X 297.0931, Y 58.0000, Z -8.0000, A 0.000, B 0.000, C 0.000 }
gfCNCPoint6[5214] = {X 297.0931, Y 58.9349, Z -8.0000, A 0.000, B 0.000, C 0.000 }
gfCNCPoint6[5215] = {X 296.9715, Y 59.9432, Z -8.0000, A 0.000, B 0.000, C 0.000 }
gfCNCPoint6[5216] = {X 296.6187, Y 60.8955, Z -8.0000, A 0.000, B 0.000, C 0.000 }
gfCNCPoint6[5217] = {X 296.0541, Y 61.7396, Z -8.0000, A 0.000, B 0.000, C 0.000 }
gfCNCPoint6[5218] = {X 295.3086, Y 62.4292, Z -8.0000, A 0.000, B 0.000, C 0.000 }
gfCNCPoint6[5219] = {X 294.4232, Y 62.9265, Z -8.0000, A 0.000, B 0.000, C 0.000 }
gfCNCPoint6[5220] = {X 293.4464, Y 63.2043, Z -8.0000, A 0.000, B 0.000, C 0.000 }
gfCNCPoint6[5221] = {X 293.3741, Y 63.2252, Z -8.0000, A 0.000, B 0.000, C 0.000 }
gfCNCPoint6[5222] = {X 293.3850, Y 92.7798, Z -8.0000, A 0.000, B 0.000, C 0.000 }
gfCNCPoint6[5223] = {X 294.2377, Y 92.9974, Z -8.0000, A 0.000, B 0.000, C 0.000 }
gfCNCPoint6[5224] = {X 295.0291, Y 93.3820, Z -8.0000, A 0.000, B 0.000, C 0.000 }
gfCNCPoint6[5225] = {X 295.7271, Y 93.9180, Z -8.0000, A 0.000, B 0.000, C 0.000 }
gfCNCPoint6[5226] = {X 296.3029, Y 94.5834, Z -8.0000, A 0.000, B 0.000, C 0.000 }
gfCNCPoint6[5227] = {X 296.7331, Y 95.3510, Z -8.0000, A 0.000, B 0.000, C 0.000 }
gfCNCPoint6[5228] = {X 297.0002, Y 96.1895, Z -8.0000, A 0.000, B 0.000, C 0.000 }
gfCNCPoint6[5229] = {X 297.0931, Y 97.0646, Z -8.0000, A 0.000, B 0.000, C 0.000 }
gfCNCPoint6[5230] = {X 297.0931, Y 98.0000, Z -8.0000, A 0.000, B 0.000, C 0.000 }
gfCNCPoint6[5231] = {X 296.9848, Y 98.9613, Z -8.0000, A 0.000, B 0.000, C 0.000 }
gfCNCPoint6[5232] = {X 296.6653, Y 99.8744, Z -8.0000, A 0.000, B 0.000, C 0.000 }
gfCNCPoint6[5233] = {X 296.1506, Y 100.6935, Z -8.0000, A 0.000, B 0.000, C 0.000 }
gfCNCPoint6[5234] = {X 295.4666, Y 101.3775, Z -8.0000, A 0.000, B 0.000, C 0.000 }
gfCNCPoint6[5235] = {X 294.6475, Y 101.8922, Z -8.0000, A 0.000, B 0.000, C 0.000 }
gfCNCPoint6[5236] = {X 293.7344, Y 102.2117, Z -8.0000, A 0.000, B 0.000, C 0.000 }
gfCNCPoint6[5237] = {X 292.7731, Y 102.3200, Z -8.0000, A 0.000, B 0.000, C 0.000 }
gfCNCPoint6[5238] = {X 276.2327, Y 102.3200, Z -8.0000, A 0.000, B 0.000, C 0.000 }
gfCNCPoint6[5239] = {X 275.2714, Y 102.2117, Z -8.0000, A 0.000, B 0.000, C 0.000 }
gfCNCPoint6[5240] = {X 274.3583, Y 101.8922, Z -8.0000, A 0.000, B 0.000, C 0.000 }
gfCNCPoint6[5241] = {X 273.5392, Y 101.3775, Z -8.0000, A 0.000, B 0.000, C 0.000 }
gfCNCPoint6[5242] = {X 272.8552, Y 100.6935, Z -8.0000, A 0.000, B 0.000, C 0.000 }
gfCNCPoint6[5243] = {X 272.3405, Y 99.8744, Z -8.0000, A 0.000, B 0.000, C 0.000 }
gfCNCPoint6[5244] = {X 272.0210, Y 98.9613, Z -8.0000, A 0.000, B 0.000, C 0.000 }
gfCNCPoint6[5245] = {X 271.9127, Y 98.0000, Z -8.0000, A 0.000, B 0.000, C 0.000 }
gfCNCPoint6[5246] = {X 271.9127, Y 97.0658, Z -8.0000, A 0.000, B 0.000, C 0.000 }
gfCNCPoint6[5247] = {X 272.0026, Y 96.1890, Z -8.0000, A 0.000, B 0.000, C 0.000 }
gfCNCPoint6[5248] = {X 272.2686, Y 95.3488, Z -8.0000, A 0.000, B 0.000, C 0.000 }
gfCNCPoint6[5249] = {X 272.6997, Y 94.5799, Z -8.0000, A 0.000, B 0.000, C 0.000 }
gfCNCPoint6[5250] = {X 273.2778, Y 93.9146, Z -8.0000, A 0.000, B 0.000, C 0.000 }
gfCNCPoint6[5251] = {X 273.9788, Y 93.3805, Z -8.0000, A 0.000, B 0.000, C 0.000 }
gfCNCPoint6[5252] = {X 274.7738, Y 92.9997, Z -8.0000, A 0.000, B 0.000, C 0.000 }
gfCNCPoint6[5253] = {X 275.6294, Y 92.7883, Z -8.0000, A 0.000, B 0.000, C 0.000 }
gfCNCPoint6[5254] = {X 275.6294, Y 85.5950, Z -8.0000, A 0.000, B 0.000, C 0.000 }
gfCNCPoint6[5255] = {X 262.6419, Y 80.5039, Z -8.0000, A 0.000, B 0.000, C 0.000 }
gfCNCPoint6[5256] = {X 237.7976, Y 96.5885, Z -8.0000, A 0.000, B 0.000, C 0.000 }
gfCNCPoint6[5257] = {X 237.7998, Y 97.0652, Z -8.0000, A 0.000, B 0.000, C 0.000 }
gfCNCPoint6[5258] = {X 237.7998, Y 98.0000, Z -8.0000, A 0.000, B 0.000, C 0.000 }
gfCNCPoint6[5259] = {X 237.6915, Y 98.9613, Z -8.0000, A 0.000, B 0.000, C 0.000 }
gfCNCPoint6[5260] = {X 237.3720, Y 99.8744, Z -8.0000, A 0.000, B 0.000, C 0.000 }
gfCNCPoint6[5261] = {X 236.8573, Y 100.6935, Z -8.0000, A 0.000, B 0.000, C 0.000 }
gfCNCPoint6[5262] = {X 236.1733, Y 101.3775, Z -8.0000, A 0.000, B 0.000, C 0.000 }
gfCNCPoint6[5263] = {X 235.3542, Y 101.8922, Z -8.0000, A 0.000, B 0.000, C 0.000 }
gfCNCPoint6[5264] = {X 234.4411, Y 102.2117, Z -8.0000, A 0.000, B 0.000, C 0.000 }
gfCNCPoint6[5265] = {X 233.4798, Y 102.3200, Z -8.0000, A 0.000, B 0.000, C 0.000 }
gfCNCPoint6[5266] = {X 214.1790, Y 102.3200, Z -8.0000, A 0.000, B 0.000, C 0.000 }
gfCNCPoint6[5267] = {X 213.7862, Y 102.3021, Z -8.0000, A 0.000, B 0.000, C 0.000 }
gfCNCPoint6[5268] = {X 213.3966, Y 102.2485, Z -8.0000, A 0.000, B 0.000, C 0.000 }
gfCNCPoint6[5269] = {X 213.0070, Y 102.3021, Z -8.0000, A 0.000, B 0.000, C 0.000 }
gfCNCPoint6[5270] = {X 212.6141, Y 102.3200, Z -8.0000, A 0.000, B 0.000, C 0.000 }
gfCNCPoint6[5271] = {X 194.9870, Y 102.3200, Z -8.0000, A 0.000, B 0.000, C 0.000 }
gfCNCPoint6[5272] = {X 194.0257, Y 102.2117, Z -8.0000, A 0.000, B 0.000, C 0.000 }
gfCNCPoint6[5273] = {X 193.1126, Y 101.8922, Z -8.0000, A 0.000, B 0.000, C 0.000 }
gfCNCPoint6[5274] = {X 192.2935, Y 101.3775, Z -8.0000, A 0.000, B 0.000, C 0.000 }
gfCNCPoint6[5275] = {X 191.6094, Y 100.6935, Z -8.0000, A 0.000, B 0.000, C 0.000 }
gfCNCPoint6[5276] = {X 191.0948, Y 99.8744, Z -8.0000, A 0.000, B 0.000, C 0.000 }
gfCNCPoint6[5277] = {X 190.7753, Y 98.9613, Z -8.0000, A 0.000, B 0.000, C 0.000 }
gfCNCPoint6[5278] = {X 190.6670, Y 98.0000, Z -8.0000, A 0.000, B 0.000, C 0.000 }
gfCNCPoint6[5279] = {X 190.6670, Y 97.0659, Z -8.0000, A 0.000, B 0.000, C 0.000 }
gfCNCPoint6[5280] = {X 190.7727, Y 96.1162, Z -8.0000, A 0.000, B 0.000, C 0.000 }
gfCNCPoint6[5281] = {X 191.0846, Y 95.2129, Z -8.0000, A 0.000, B 0.000, C 0.000 }
gfCNCPoint6[5282] = {X 191.5874, Y 94.4003, Z -8.0000, A 0.000, B 0.000, C 0.000 }
gfCNCPoint6[5283] = {X 188.5647, Y 91.1002, Z -8.0000, A 0.000, B 0.000, C 0.000 }
gfCNCPoint6[5284] = {X 150.0898, Y 91.1002, Z -8.0000, A 0.000, B 0.000, C 0.000 }
gfCNCPoint6[5285] = {X 147.1458, Y 94.3619, Z -8.0000, A 0.000, B 0.000, C 0.000 }
gfCNCPoint6[5286] = {X 147.6651, Y 95.1833, Z -8.0000, A 0.000, B 0.000, C 0.000 }
gfCNCPoint6[5287] = {X 147.9883, Y 96.0999, Z -8.0000, A 0.000, B 0.000, C 0.000 }
gfCNCPoint6[5288] = {X 148.0991, Y 97.0654, Z -8.0000, A 0.000, B 0.000, C 0.000 }
gfCNCPoint6[5289] = {X 148.0991, Y 98.0000, Z -8.0000, A 0.000, B 0.000, C 0.000 }
gfCNCPoint6[5290] = {X 147.9908, Y 98.9613, Z -8.0000, A 0.000, B 0.000, C 0.000 }
gfCNCPoint6[5291] = {X 147.6713, Y 99.8744, Z -8.0000, A 0.000, B 0.000, C 0.000 }
gfCNCPoint6[5292] = {X 147.1566, Y 100.6935, Z -8.0000, A 0.000, B 0.000, C 0.000 }
gfCNCPoint6[5293] = {X 146.4726, Y 101.3775, Z -8.0000, A 0.000, B 0.000, C 0.000 }
gfCNCPoint6[5294] = {X 145.6535, Y 101.8922, Z -8.0000, A 0.000, B 0.000, C 0.000 }
gfCNCPoint6[5295] = {X 144.7404, Y 102.2117, Z -8.0000, A 0.000, B 0.000, C 0.000 }
gfCNCPoint6[5296] = {X 143.7791, Y 102.3200, Z -8.0000, A 0.000, B 0.000, C 0.000 }
gfCNCPoint6[5297] = {X 125.0000, Y 102.3200, Z -8.0000, A 0.000, B 0.000, C 0.000 }
gfCNCPoint6[5298] = {X 124.0387, Y 102.2117, Z -8.0000, A 0.000, B 0.000, C 0.000 }
gfCNCPoint6[5299] = {X 123.1256, Y 101.8922, Z -8.0000, A 0.000, B 0.000, C 0.000 }
gfCNCPoint6[5300] = {X 122.3065, Y 101.3775, Z -8.0000, A 0.000, B 0.000, C 0.000 }
gfCNCPoint6[5301] = {X 121.6225, Y 100.6935, Z -8.0000, A 0.000, B 0.000, C 0.000 }
gfCNCPoint6[5302] = {X 121.1078, Y 99.8744, Z -8.0000, A 0.000, B 0.000, C 0.000 }
gfCNCPoint6[5303] = {X 120.7883, Y 98.9613, Z -8.0000, A 0.000, B 0.000, C 0.000 }
gfCNCPoint6[5304] = {X 120.6800, Y 98.0000, Z -8.0000, A 0.000, B 0.000, C 0.000 }
gfCNCPoint6[5305] = {X 120.6800, Y 97.0659, Z -8.0000, A 0.000, B 0.000, C 0.000 }
gfCNCPoint6[5306] = {X 120.7831, Y 96.1278, Z -8.0000, A 0.000, B 0.000, C 0.000 }
gfCNCPoint6[5307] = {X 121.0875, Y 95.2344, Z -8.0000, A 0.000, B 0.000, C 0.000 }
gfCNCPoint6[5308] = {X 121.5786, Y 94.4284, Z -8.0000, A 0.000, B 0.000, C 0.000 }
gfCNCPoint6[5309] = {X 122.2331, Y 93.7483, Z -8.0000, A 0.000, B 0.000, C 0.000 }
gfCNCPoint6[5310] = {X 123.0196, Y 93.2266, Z -8.0000, A 0.000, B 0.000, C 0.000 }
gfCNCPoint6[5311] = {X 123.9007, Y 92.8882, Z -8.0000, A 0.000, B 0.000, C 0.000 }
gfCNCPoint6[5312] = {X 124.8342, Y 92.7491, Z -8.0000, A 0.000, B 0.000, C 0.000 }
gfCNCPoint6[5313] = {X 124.8798, Y 92.7310, Z -8.0000, A 0.000, B 0.000, C 0.000 }
gfCNCPoint6[5314] = {X 124.9277, Y 92.7201, Z -8.0000, A 0.000, B 0.000, C 0.000 }
gfCNCPoint6[5315] = {X 125.4493, Y 92.6428, Z -8.0000, A 0.000, B 0.000, C 0.000 }
gfCNCPoint6[5316] = {X 126.2803, Y 92.5026, Z -8.0000, A 0.000, B 0.000, C 0.000 }
gfCNCPoint6[5317] = {X 127.0999, Y 92.3065, Z -8.0000, A 0.000, B 0.000, C 0.000 }
gfCNCPoint6[5318] = {X 128.2870, Y 91.1904, Z -8.0000, A 0.000, B 0.000, C 0.000 }
gfCNCPoint6[5319] = {X 129.4114, Y 90.0111, Z -8.0000, A 0.000, B 0.000, C 0.000 }
gfCNCPoint6[5320] = {X 140.6793, Y 77.6382, Z -8.0000, A 0.000, B 0.000, C 0.000 }
gfCNCPoint6[5321] = {X 137.7219, Y 74.9449, Z -8.0000, A 0.000, B 0.000, C 0.000 }
gfCNCPoint6[5322] = {X 140.7385, Y 77.6921, Z -8.0000, A 0.000, B 0.000, C 0.000 }
gfCNCPoint6[5323] = {X 155.7321, Y 61.2281, Z -8.0000, A 0.000, B 0.000, C 0.000 }
gfCNCPoint6[5324] = {X 155.3665, Y 60.5220, Z -8.0000, A 0.000, B 0.000, C 0.000 }
gfCNCPoint6[5325] = {X 155.1392, Y 59.7601, Z -8.0000, A 0.000, B 0.000, C 0.000 }
gfCNCPoint6[5326] = {X 155.0581, Y 58.9691, Z -8.0000, A 0.000, B 0.000, C 0.000 }
gfCNCPoint6[5327] = {X 155.0580, Y 58.0000, Z -8.0000, A 0.000, B 0.000, C 0.000 }
gfCNCPoint6[5328] = {X 155.1643, Y 57.0565, Z -8.0000, A 0.000, B 0.000, C 0.000 }
gfCNCPoint6[5329] = {X 155.4778, Y 56.1603, Z -8.0000, A 0.000, B 0.000, C 0.000 }
gfCNCPoint6[5330] = {X 155.9830, Y 55.3564, Z -8.0000, A 0.000, B 0.000, C 0.000 }
gfCNCPoint6[5331] = {X 156.6544, Y 54.6850, Z -8.0000, A 0.000, B 0.000, C 0.000 }
gfCNCPoint6[5332] = {X 157.4583, Y 54.1799, Z -8.0000, A 0.000, B 0.000, C 0.000 }
gfCNCPoint6[5333] = {X 158.3545, Y 53.8663, Z -8.0000, A 0.000, B 0.000, C 0.000 }
gfCNCPoint6[5334] = {X 159.2980, Y 53.7600, Z -8.0000, A 0.000, B 0.000, C 0.000 }
gfCNCPoint6[5335] = {X 178.5335, Y 53.7600, Z -8.0000, A 0.000, B 0.000, C 0.000 }
gfCNCPoint6[5336] = {X 179.4770, Y 53.8663, Z -8.0000, A 0.000, B 0.000, C 0.000 }
gfCNCPoint6[5337] = {X 180.3732, Y 54.1799, Z -8.0000, A 0.000, B 0.000, C 0.000 }
gfCNCPoint6[5338] = {X 181.1771, Y 54.6850, Z -8.0000, A 0.000, B 0.000, C 0.000 }
gfCNCPoint6[5339] = {X 181.8485, Y 55.3564, Z -8.0000, A 0.000, B 0.000, C 0.000 }
gfCNCPoint6[5340] = {X 182.3536, Y 56.1603, Z -8.0000, A 0.000, B 0.000, C 0.000 }
gfCNCPoint6[5341] = {X 182.6672, Y 57.0565, Z -8.0000, A 0.000, B 0.000, C 0.000 }
gfCNCPoint6[5342] = {X 182.7735, Y 58.0000, Z -8.0000, A 0.000, B 0.000, C 0.000 }
gfCNCPoint6[5343] = {X 182.7735, Y 58.9342, Z -8.0000, A 0.000, B 0.000, C 0.000 }
gfCNCPoint6[5344] = {X 182.6985, Y 59.7281, Z -8.0000, A 0.000, B 0.000, C 0.000 }
gfCNCPoint6[5345] = {X 182.4762, Y 60.4938, Z -8.0000, A 0.000, B 0.000, C 0.000 }
gfCNCPoint6[5346] = {X 182.1145, Y 61.2044, Z -8.0000, A 0.000, B 0.000, C 0.000 }
gfCNCPoint6[5347] = {X 209.2352, Y 90.8109, Z -8.0000, A 0.000, B 0.000, C 0.000 }
gfCNCPoint6[5348] = {X 209.9099, Y 91.5098, Z -8.0000, A 0.000, B 0.000, C 0.000 }
gfCNCPoint6[5349] = {X 210.6203, Y 92.1725, Z -8.0000, A 0.000, B 0.000, C 0.000 }
gfCNCPoint6[5350] = {X 211.0329, Y 92.4517, Z -8.0000, A 0.000, B 0.000, C 0.000 }
gfCNCPoint6[5351] = {X 211.5033, Y 92.6159, Z -8.0000, A 0.000, B 0.000, C 0.000 }
gfCNCPoint6[5352] = {X 212.0942, Y 92.7396, Z -8.0000, A 0.000, B 0.000, C 0.000 }
gfCNCPoint6[5353] = {X 213.3852, Y 92.9000, Z -8.0000, A 0.000, B 0.000, C 0.000 }
gfCNCPoint6[5354] = {X 214.4465, Y 92.8157, Z -8.0000, A 0.000, B 0.000, C 0.000 }
gfCNCPoint6[5355] = {X 215.5093, Y 92.7542, Z -8.0000, A 0.000, B 0.000, C 0.000 }
gfCNCPoint6[5356] = {X 216.1939, Y 92.6796, Z -8.0000, A 0.000, B 0.000, C 0.000 }
gfCNCPoint6[5357] = {X 216.8530, Y 92.4802, Z -8.0000, A 0.000, B 0.000, C 0.000 }
gfCNCPoint6[5358] = {X 217.4643, Y 92.1630, Z -8.0000, A 0.000, B 0.000, C 0.000 }
gfCNCPoint6[5359] = {X 223.0046, Y 88.5876, Z -8.0000, A 0.000, B 0.000, C 0.000 }
gfCNCPoint6[5360] = {X 246.0021, Y 73.8825, Z -8.0000, A 0.000, B 0.000, C 0.000 }
gfCNCPoint6[5361] = {X 221.6603, Y 64.3308, Z -8.0000, A 0.000, B 0.000, C 0.000 }
gfCNCPoint6[5362] = {X 219.8841, Y 63.7365, Z -8.0000, A 0.000, B 0.000, C 0.000 }
gfCNCPoint6[5363] = {X 218.0517, Y 63.3484, Z -8.0000, A 0.000, B 0.000, C 0.000 }
gfCNCPoint6[5364] = {X 216.1871, Y 63.1716, Z -8.0000, A 0.000, B 0.000, C 0.000 }
gfCNCPoint6[5365] = {X 215.2724, Y 63.0398, Z -8.0000, A 0.000, B 0.000, C 0.000 }
gfCNCPoint6[5366] = {X 214.4081, Y 62.7131, Z -8.0000, A 0.000, B 0.000, C 0.000 }
gfCNCPoint6[5367] = {X 213.6351, Y 62.2068, Z -8.0000, A 0.000, B 0.000, C 0.000 }
gfCNCPoint6[5368] = {X 212.9901, Y 61.5450, Z -8.0000, A 0.000, B 0.000, C 0.000 }
gfCNCPoint6[5369] = {X 212.5038, Y 60.7592, Z -8.0000, A 0.000, B 0.000, C 0.000 }
gfCNCPoint6[5370] = {X 212.1992, Y 59.8868, Z -8.0000, A 0.000, B 0.000, C 0.000 }
gfCNCPoint6[5371] = {X 212.0910, Y 58.9691, Z -8.0000, A 0.000, B 0.000, C 0.000 }
gfCNCPoint6[5372] = {X 212.0908, Y 58.0000, Z -8.0000, A 0.000, B 0.000, C 0.000 }
gfCNCPoint6[5373] = {X 212.1971, Y 57.0565, Z -8.0000, A 0.000, B 0.000, C 0.000 }
gfCNCPoint6[5374] = {X 212.5107, Y 56.1603, Z -8.0000, A 0.000, B 0.000, C 0.000 }
gfCNCPoint6[5375] = {X 213.0158, Y 55.3564, Z -8.0000, A 0.000, B 0.000, C 0.000 }
gfCNCPoint6[5376] = {X 213.6872, Y 54.6850, Z -8.0000, A 0.000, B 0.000, C 0.000 }
gfCNCPoint6[5377] = {X 214.4911, Y 54.1799, Z -8.0000, A 0.000, B 0.000, C 0.000 }
gfCNCPoint6[5378] = {X 215.3873, Y 53.8663, Z -8.0000, A 0.000, B 0.000, C 0.000 }
gfCNCPoint6[5379] = {X 216.3308, Y 53.7600, Z -8.0000, A 0.000, B 0.000, C 0.000 }
gfCNCPoint6[5380] = {X 237.2617, Y 53.7600, Z -8.0000, A 0.000, B 0.000, C 0.000 }
gfCNCPoint6[5381] = {X 238.2052, Y 53.8663, Z -8.0000, A 0.000, B 0.000, C 0.000 }
gfCNCPoint6[5382] = {X 239.1014, Y 54.1799, Z -8.0000, A 0.000, B 0.000, C 0.000 }
gfCNCPoint6[5383] = {X 239.9053, Y 54.6850, Z -8.0000, A 0.000, B 0.000, C 0.000 }
gfCNCPoint6[5384] = {X 240.5767, Y 55.3564, Z -8.0000, A 0.000, B 0.000, C 0.000 }
gfCNCPoint6[5385] = {X 241.0818, Y 56.1603, Z -8.0000, A 0.000, B 0.000, C 0.000 }
gfCNCPoint6[5386] = {X 241.3954, Y 57.0565, Z -8.0000, A 0.000, B 0.000, C 0.000 }
gfCNCPoint6[5387] = {X 241.5017, Y 58.0000, Z -8.0000, A 0.000, B 0.000, C 0.000 }
gfCNCPoint6[5388] = {X 241.5017, Y 58.2862, Z -8.0000, A 0.000, B 0.000, C 0.000 }
gfCNCPoint6[5389] = {X 248.0859, Y 60.8537, Z -8.0000, A 0.000, B 0.000, C 0.000 }
gfCNCPoint6[5390] = {X 275.7115, Y 71.8189, Z -8.0000, A 0.000, B 0.000, C 0.000 }
gfCNCPoint6[5391] = {X 275.7133, Y 63.1421, Z -8.0000, A 0.000, B 0.000, C 0.000 }
gfCNCPoint6[5392] = {X 274.8649, Y 62.9474, Z -8.0000, A 0.000, B 0.000, C 0.000 }
gfCNCPoint6[5393] = {X 274.0740, Y 62.5834, Z -8.0000, A 0.000, B 0.000, C 0.000 }
gfCNCPoint6[5394] = {X 273.3742, Y 62.0657, Z -8.0000, A 0.000, B 0.000, C 0.000 }
gfCNCPoint6[5395] = {X 272.7949, Y 61.4159, Z -8.0000, A 0.000, B 0.000, C 0.000 }
gfCNCPoint6[5396] = {X 272.3605, Y 60.6615, Z -8.0000, A 0.000, B 0.000, C 0.000 }
gfCNCPoint6[5397] = {X 272.0893, Y 59.8342, Z -8.0000, A 0.000, B 0.000, C 0.000 }
gfCNCPoint6[5398] = {X 271.9928, Y 58.9691, Z -8.0000, A 0.000, B 0.000, C 0.000 }
gfCNCPoint6[5399] = {X 271.9927, Y 58.0000, Z -8.0000, A 0.000, B 0.000, C 0.000 }
gfCNCPoint6[5400] = {X 272.0990, Y 57.0565, Z -8.0000, A 0.000, B 0.000, C 0.000 }
gfCNCPoint6[5401] = {X 272.4126, Y 56.1603, Z -8.0000, A 0.000, B 0.000, C 0.000 }
gfCNCPoint6[5402] = {X 272.9177, Y 55.3564, Z -8.0000, A 0.000, B 0.000, C 0.000 }
gfCNCPoint6[5403] = {X 273.5891, Y 54.6850, Z -8.0000, A 0.000, B 0.000, C 0.000 }
gfCNCPoint6[5404] = {X 274.3930, Y 54.1799, Z -8.0000, A 0.000, B 0.000, C 0.000 }
gfCNCPoint6[5405] = {X 275.2892, Y 53.8663, Z -8.0000, A 0.000, B 0.000, C 0.000 }
gfCNCPoint6[5406] = {X 276.2327, Y 53.7600, Z -8.0000, A 0.000, B 0.000, C 0.000 }
gfCNCPoint6[5407] = {X 292.7731, Y 53.7600, Z -8.0000, A 0.000, B 0.000, C 0.000 }
gfCNCPoint6[5408] = {X 293.7166, Y 53.8663, Z -8.0000, A 0.000, B 0.000, C 0.000 }
gfCNCPoint6[5409] = {X 294.6128, Y 54.1799, Z -8.0000, A 0.000, B 0.000, C 0.000 }
gfCNCPoint6[5410] = {X 295.4167, Y 54.6850, Z -8.0000, A 0.000, B 0.000, C 0.000 }
gfCNCPoint6[5411] = {X 296.0881, Y 55.3564, Z -8.0000, A 0.000, B 0.000, C 0.000 }
gfCNCPoint6[5412] = {X 296.5932, Y 56.1603, Z -8.0000, A 0.000, B 0.000, C 0.000 }
gfCNCPoint6[5413] = {X 296.9068, Y 57.0565, Z -8.0000, A 0.000, B 0.000, C 0.000 }
gfCNCPoint6[5414] = {X 297.0131, Y 58.0000, Z -8.0000, A 0.000, B 0.000, C 0.000 }
gfCNCPoint6[5415] = {X 297.0131, Y 58.9347, Z -8.0000, A 0.000, B 0.000, C 0.000 }
gfCNCPoint6[5416] = {X 296.8935, Y 59.9251, Z -8.0000, A 0.000, B 0.000, C 0.000 }
gfCNCPoint6[5417] = {X 296.5467, Y 60.8605, Z -8.0000, A 0.000, B 0.000, C 0.000 }
gfCNCPoint6[5418] = {X 295.9917, Y 61.6895, Z -8.0000, A 0.000, B 0.000, C 0.000 }
gfCNCPoint6[5419] = {X 295.2589, Y 62.3664, Z -8.0000, A 0.000, B 0.000, C 0.000 }
gfCNCPoint6[5420] = {X 294.3887, Y 62.8542, Z -8.0000, A 0.000, B 0.000, C 0.000 }
gfCNCPoint6[5421] = {X 293.4288, Y 63.1260, Z -8.0000, A 0.000, B 0.000, C 0.000 }
gfCNCPoint6[5422] = {X 293.2941, Y 63.1651, Z -8.0000, A 0.000, B 0.000, C 0.000 }
gfCNCPoint6[5423] = {X 293.3050, Y 92.8493, Z -8.0000, A 0.000, B 0.000, C 0.000 }
gfCNCPoint6[5424] = {X 294.1546, Y 93.0526, Z -8.0000, A 0.000, B 0.000, C 0.000 }
gfCNCPoint6[5425] = {X 294.9451, Y 93.4245, Z -8.0000, A 0.000, B 0.000, C 0.000 }
gfCNCPoint6[5426] = {X 295.6434, Y 93.9493, Z -8.0000, A 0.000, B 0.000, C 0.000 }
gfCNCPoint6[5427] = {X 296.2204, Y 94.6053, Z -8.0000, A 0.000, B 0.000, C 0.000 }
gfCNCPoint6[5428] = {X 296.6519, Y 95.3649, Z -8.0000, A 0.000, B 0.000, C 0.000 }
gfCNCPoint6[5429] = {X 296.9198, Y 96.1963, Z -8.0000, A 0.000, B 0.000, C 0.000 }
gfCNCPoint6[5430] = {X 297.0131, Y 97.0649, Z -8.0000, A 0.000, B 0.000, C 0.000 }
gfCNCPoint6[5431] = {X 297.0131, Y 98.0000, Z -8.0000, A 0.000, B 0.000, C 0.000 }
gfCNCPoint6[5432] = {X 296.9068, Y 98.9435, Z -8.0000, A 0.000, B 0.000, C 0.000 }
gfCNCPoint6[5433] = {X 296.5932, Y 99.8397, Z -8.0000, A 0.000, B 0.000, C 0.000 }
gfCNCPoint6[5434] = {X 296.0881, Y 100.6436, Z -8.0000, A 0.000, B 0.000, C 0.000 }
gfCNCPoint6[5435] = {X 295.4167, Y 101.3150, Z -8.0000, A 0.000, B 0.000, C 0.000 }
gfCNCPoint6[5436] = {X 294.6128, Y 101.8201, Z -8.0000, A 0.000, B 0.000, C 0.000 }
gfCNCPoint6[5437] = {X 293.7166, Y 102.1337, Z -8.0000, A 0.000, B 0.000, C 0.000 }
gfCNCPoint6[5438] = {X 292.7731, Y 102.2400, Z -8.0000, A 0.000, B 0.000, C 0.000 }
gfCNCPoint6[5439] = {X 276.2327, Y 102.2400, Z -8.0000, A 0.000, B 0.000, C 0.000 }
gfCNCPoint6[5440] = {X 275.2892, Y 102.1337, Z -8.0000, A 0.000, B 0.000, C 0.000 }
gfCNCPoint6[5441] = {X 274.3930, Y 101.8201, Z -8.0000, A 0.000, B 0.000, C 0.000 }
gfCNCPoint6[5442] = {X 273.5891, Y 101.3150, Z -8.0000, A 0.000, B 0.000, C 0.000 }
gfCNCPoint6[5443] = {X 272.9177, Y 100.6436, Z -8.0000, A 0.000, B 0.000, C 0.000 }
gfCNCPoint6[5444] = {X 272.4126, Y 99.8397, Z -8.0000, A 0.000, B 0.000, C 0.000 }
gfCNCPoint6[5445] = {X 272.0990, Y 98.9435, Z -8.0000, A 0.000, B 0.000, C 0.000 }
gfCNCPoint6[5446] = {X 271.9927, Y 98.0000, Z -8.0000, A 0.000, B 0.000, C 0.000 }
gfCNCPoint6[5447] = {X 271.9927, Y 97.0658, Z -8.0000, A 0.000, B 0.000, C 0.000 }
gfCNCPoint6[5448] = {X 272.0830, Y 96.1956, Z -8.0000, A 0.000, B 0.000, C 0.000 }
gfCNCPoint6[5449] = {X 272.3500, Y 95.3624, Z -8.0000, A 0.000, B 0.000, C 0.000 }
gfCNCPoint6[5450] = {X 272.7823, Y 94.6017, Z -8.0000, A 0.000, B 0.000, C 0.000 }
gfCNCPoint6[5451] = {X 273.3615, Y 93.9460, Z -8.0000, A 0.000, B 0.000, C 0.000 }
gfCNCPoint6[5452] = {X 274.0630, Y 93.4231, Z -8.0000, A 0.000, B 0.000, C 0.000 }
gfCNCPoint6[5453] = {X 274.8569, Y 93.0553, Z -8.0000, A 0.000, B 0.000, C 0.000 }
gfCNCPoint6[5454] = {X 275.7094, Y 92.8584, Z -8.0000, A 0.000, B 0.000, C 0.000 }
gfCNCPoint6[5455] = {X 275.7094, Y 85.5404, Z -8.0000, A 0.000, B 0.000, C 0.000 }
gfCNCPoint6[5456] = {X 262.6329, Y 80.4144, Z -8.0000, A 0.000, B 0.000, C 0.000 }
gfCNCPoint6[5457] = {X 237.7174, Y 96.5451, Z -8.0000, A 0.000, B 0.000, C 0.000 }
gfCNCPoint6[5458] = {X 237.7198, Y 97.0654, Z -8.0000, A 0.000, B 0.000, C 0.000 }
gfCNCPoint6[5459] = {X 237.7198, Y 98.0000, Z -8.0000, A 0.000, B 0.000, C 0.000 }
gfCNCPoint6[5460] = {X 237.6135, Y 98.9435, Z -8.0000, A 0.000, B 0.000, C 0.000 }
gfCNCPoint6[5461] = {X 237.2999, Y 99.8397, Z -8.0000, A 0.000, B 0.000, C 0.000 }
gfCNCPoint6[5462] = {X 236.7948, Y 100.6436, Z -8.0000, A 0.000, B 0.000, C 0.000 }
gfCNCPoint6[5463] = {X 236.1234, Y 101.3150, Z -8.0000, A 0.000, B 0.000, C 0.000 }
gfCNCPoint6[5464] = {X 235.3195, Y 101.8201, Z -8.0000, A 0.000, B 0.000, C 0.000 }
gfCNCPoint6[5465] = {X 234.4233, Y 102.1337, Z -8.0000, A 0.000, B 0.000, C 0.000 }
gfCNCPoint6[5466] = {X 233.4798, Y 102.2400, Z -8.0000, A 0.000, B 0.000, C 0.000 }
gfCNCPoint6[5467] = {X 214.1790, Y 102.2400, Z -8.0000, A 0.000, B 0.000, C 0.000 }
gfCNCPoint6[5468] = {X 213.7861, Y 102.2218, Z -8.0000, A 0.000, B 0.000, C 0.000 }
gfCNCPoint6[5469] = {X 213.3966, Y 102.1672, Z -8.0000, A 0.000, B 0.000, C 0.000 }
gfCNCPoint6[5470] = {X 213.0070, Y 102.2218, Z -8.0000, A 0.000, B 0.000, C 0.000 }
gfCNCPoint6[5471] = {X 212.6141, Y 102.2400, Z -8.0000, A 0.000, B 0.000, C 0.000 }
gfCNCPoint6[5472] = {X 194.9870, Y 102.2400, Z -8.0000, A 0.000, B 0.000, C 0.000 }
gfCNCPoint6[5473] = {X 194.0435, Y 102.1337, Z -8.0000, A 0.000, B 0.000, C 0.000 }
gfCNCPoint6[5474] = {X 193.1473, Y 101.8201, Z -8.0000, A 0.000, B 0.000, C 0.000 }
gfCNCPoint6[5475] = {X 192.3434, Y 101.3150, Z -8.0000, A 0.000, B 0.000, C 0.000 }
gfCNCPoint6[5476] = {X 191.6720, Y 100.6436, Z -8.0000, A 0.000, B 0.000, C 0.000 }
gfCNCPoint6[5477] = {X 191.1669, Y 99.8397, Z -8.0000, A 0.000, B 0.000, C 0.000 }
gfCNCPoint6[5478] = {X 190.8533, Y 98.9435, Z -8.0000, A 0.000, B 0.000, C 0.000 }
gfCNCPoint6[5479] = {X 190.7470, Y 98.0000, Z -8.0000, A 0.000, B 0.000, C 0.000 }
gfCNCPoint6[5480] = {X 190.7470, Y 97.0659, Z -8.0000, A 0.000, B 0.000, C 0.000 }
gfCNCPoint6[5481] = {X 190.8557, Y 96.1118, Z -8.0000, A 0.000, B 0.000, C 0.000 }
gfCNCPoint6[5482] = {X 191.1764, Y 95.2065, Z -8.0000, A 0.000, B 0.000, C 0.000 }
gfCNCPoint6[5483] = {X 191.6926, Y 94.3967, Z -8.0000, A 0.000, B 0.000, C 0.000 }
gfCNCPoint6[5484] = {X 188.5999, Y 91.0202, Z -8.0000, A 0.000, B 0.000, C 0.000 }
gfCNCPoint6[5485] = {X 150.0543, Y 91.0202, Z -8.0000, A 0.000, B 0.000, C 0.000 }
gfCNCPoint6[5486] = {X 147.0404, Y 94.3592, Z -8.0000, A 0.000, B 0.000, C 0.000 }
gfCNCPoint6[5487] = {X 147.5731, Y 95.1775, Z -8.0000, A 0.000, B 0.000, C 0.000 }
gfCNCPoint6[5488] = {X 147.9052, Y 96.0958, Z -8.0000, A 0.000, B 0.000, C 0.000 }
gfCNCPoint6[5489] = {X 148.0191, Y 97.0656, Z -8.0000, A 0.000, B 0.000, C 0.000 }
gfCNCPoint6[5490] = {X 148.0191, Y 98.0000, Z -8.0000, A 0.000, B 0.000, C 0.000 }
gfCNCPoint6[5491] = {X 147.9128, Y 98.9435, Z -8.0000, A 0.000, B 0.000, C 0.000 }
gfCNCPoint6[5492] = {X 147.5992, Y 99.8397, Z -8.0000, A 0.000, B 0.000, C 0.000 }
gfCNCPoint6[5493] = {X 147.0941, Y 100.6436, Z -8.0000, A 0.000, B 0.000, C 0.000 }
gfCNCPoint6[5494] = {X 146.4227, Y 101.3150, Z -8.0000, A 0.000, B 0.000, C 0.000 }
gfCNCPoint6[5495] = {X 145.6188, Y 101.8201, Z -8.0000, A 0.000, B 0.000, C 0.000 }
gfCNCPoint6[5496] = {X 144.7226, Y 102.1337, Z -8.0000, A 0.000, B 0.000, C 0.000 }
gfCNCPoint6[5497] = {X 143.7791, Y 102.2400, Z -8.0000, A 0.000, B 0.000, C 0.000 }
gfCNCPoint6[5498] = {X 125.0000, Y 102.2400, Z -8.0000, A 0.000, B 0.000, C 0.000 }
gfCNCPoint6[5499] = {X 124.0565, Y 102.1337, Z -8.0000, A 0.000, B 0.000, C 0.000 }
gfCNCPoint6[5500] = {X 123.1603, Y 101.8201, Z -8.0000, A 0.000, B 0.000, C 0.000 }
gfCNCPoint6[5501] = {X 122.3564, Y 101.3150, Z -8.0000, A 0.000, B 0.000, C 0.000 }
gfCNCPoint6[5502] = {X 121.6850, Y 100.6436, Z -8.0000, A 0.000, B 0.000, C 0.000 }
gfCNCPoint6[5503] = {X 121.1799, Y 99.8397, Z -8.0000, A 0.000, B 0.000, C 0.000 }
gfCNCPoint6[5504] = {X 120.8663, Y 98.9435, Z -8.0000, A 0.000, B 0.000, C 0.000 }
gfCNCPoint6[5505] = {X 120.7600, Y 98.0000, Z -8.0000, A 0.000, B 0.000, C 0.000 }
gfCNCPoint6[5506] = {X 120.7600, Y 97.0659, Z -8.0000, A 0.000, B 0.000, C 0.000 }
gfCNCPoint6[5507] = {X 120.8618, Y 96.1426, Z -8.0000, A 0.000, B 0.000, C 0.000 }
gfCNCPoint6[5508] = {X 121.1621, Y 95.2636, Z -8.0000, A 0.000, B 0.000, C 0.000 }
gfCNCPoint6[5509] = {X 121.6467, Y 94.4711, Z -8.0000, A 0.000, B 0.000, C 0.000 }
gfCNCPoint6[5510] = {X 122.2923, Y 93.8032, Z -8.0000, A 0.000, B 0.000, C 0.000 }
gfCNCPoint6[5511] = {X 123.0678, Y 93.2918, Z -8.0000, A 0.000, B 0.000, C 0.000 }
gfCNCPoint6[5512] = {X 123.9360, Y 92.9616, Z -8.0000, A 0.000, B 0.000, C 0.000 }
gfCNCPoint6[5513] = {X 124.8553, Y 92.8284, Z -8.0000, A 0.000, B 0.000, C 0.000 }
gfCNCPoint6[5514] = {X 124.8960, Y 92.8099, Z -8.0000, A 0.000, B 0.000, C 0.000 }
gfCNCPoint6[5515] = {X 124.9394, Y 92.7993, Z -8.0000, A 0.000, B 0.000, C 0.000 }
gfCNCPoint6[5516] = {X 125.4605, Y 92.7220, Z -8.0000, A 0.000, B 0.000, C 0.000 }
gfCNCPoint6[5517] = {X 126.3057, Y 92.5790, Z -8.0000, A 0.000, B 0.000, C 0.000 }
gfCNCPoint6[5518] = {X 127.1391, Y 92.3786, Z -8.0000, A 0.000, B 0.000, C 0.000 }
gfCNCPoint6[5519] = {X 128.3368, Y 91.2538, Z -8.0000, A 0.000, B 0.000, C 0.000 }
gfCNCPoint6[5520] = {X 129.4708, Y 90.0647, Z -8.0000, A 0.000, B 0.000, C 0.000 }
gfCNCPoint6[5521] = {X 140.7385, Y 77.6921, Z -8.0000, A 0.000, B 0.000, C 0.000 }
gfCNCPoint6[5522] = {X 137.7811, Y 74.9988, Z -8.0000, A 0.000, B 0.000, C 0.000 }
gfCNCPoint6[5523] = {X 140.7976, Y 77.7459, Z -8.0000, A 0.000, B 0.000, C 0.000 }
gfCNCPoint6[5524] = {X 155.8330, Y 61.2361, Z -8.0000, A 0.000, B 0.000, C 0.000 }
gfCNCPoint6[5525] = {X 155.4562, Y 60.5299, Z -8.0000, A 0.000, B 0.000, C 0.000 }
gfCNCPoint6[5526] = {X 155.2217, Y 59.7645, Z -8.0000, A 0.000, B 0.000, C 0.000 }
gfCNCPoint6[5527] = {X 155.1381, Y 58.9684, Z -8.0000, A 0.000, B 0.000, C 0.000 }
gfCNCPoint6[5528] = {X 155.1380, Y 58.0000, Z -8.0000, A 0.000, B 0.000, C 0.000 }
gfCNCPoint6[5529] = {X 155.2423, Y 57.0743, Z -8.0000, A 0.000, B 0.000, C 0.000 }
gfCNCPoint6[5530] = {X 155.5499, Y 56.1950, Z -8.0000, A 0.000, B 0.000, C 0.000 }
gfCNCPoint6[5531] = {X 156.0455, Y 55.4063, Z -8.0000, A 0.000, B 0.000, C 0.000 }
gfCNCPoint6[5532] = {X 156.7042, Y 54.7476, Z -8.0000, A 0.000, B 0.000, C 0.000 }
gfCNCPoint6[5533] = {X 157.4930, Y 54.2520, Z -8.0000, A 0.000, B 0.000, C 0.000 }
gfCNCPoint6[5534] = {X 158.3723, Y 53.9443, Z -8.0000, A 0.000, B 0.000, C 0.000 }
gfCNCPoint6[5535] = {X 159.2980, Y 53.8400, Z -8.0000, A 0.000, B 0.000, C 0.000 }
gfCNCPoint6[5536] = {X 178.5335, Y 53.8400, Z -8.0000, A 0.000, B 0.000, C 0.000 }
gfCNCPoint6[5537] = {X 179.4592, Y 53.9443, Z -8.0000, A 0.000, B 0.000, C 0.000 }
gfCNCPoint6[5538] = {X 180.3385, Y 54.2520, Z -8.0000, A 0.000, B 0.000, C 0.000 }
gfCNCPoint6[5539] = {X 181.1272, Y 54.7476, Z -8.0000, A 0.000, B 0.000, C 0.000 }
gfCNCPoint6[5540] = {X 181.7859, Y 55.4063, Z -8.0000, A 0.000, B 0.000, C 0.000 }
gfCNCPoint6[5541] = {X 182.2815, Y 56.1950, Z -8.0000, A 0.000, B 0.000, C 0.000 }
gfCNCPoint6[5542] = {X 182.5892, Y 57.0743, Z -8.0000, A 0.000, B 0.000, C 0.000 }
gfCNCPoint6[5543] = {X 182.6935, Y 58.0000, Z -8.0000, A 0.000, B 0.000, C 0.000 }
gfCNCPoint6[5544] = {X 182.6935, Y 58.9342, Z -8.0000, A 0.000, B 0.000, C 0.000 }
gfCNCPoint6[5545] = {X 182.6160, Y 59.7331, Z -8.0000, A 0.000, B 0.000, C 0.000 }
gfCNCPoint6[5546] = {X 182.3866, Y 60.5022, Z -8.0000, A 0.000, B 0.000, C 0.000 }
gfCNCPoint6[5547] = {X 182.0138, Y 61.2129, Z -8.0000, A 0.000, B 0.000, C 0.000 }
gfCNCPoint6[5548] = {X 209.1762, Y 90.8649, Z -8.0000, A 0.000, B 0.000, C 0.000 }
gfCNCPoint6[5549] = {X 209.8538, Y 91.5669, Z -8.0000, A 0.000, B 0.000, C 0.000 }
gfCNCPoint6[5550] = {X 210.5673, Y 92.2324, Z -8.0000, A 0.000, B 0.000, C 0.000 }
gfCNCPoint6[5551] = {X 210.9970, Y 92.5232, Z -8.0000, A 0.000, B 0.000, C 0.000 }
gfCNCPoint6[5552] = {X 211.4869, Y 92.6942, Z -8.0000, A 0.000, B 0.000, C 0.000 }
gfCNCPoint6[5553] = {X 212.0810, Y 92.8186, Z -8.0000, A 0.000, B 0.000, C 0.000 }
gfCNCPoint6[5554] = {X 213.3851, Y 92.9829, Z -8.0000, A 0.000, B 0.000, C 0.000 }
gfCNCPoint6[5555] = {X 213.3992, Y 92.9791, Z -8.0000, A 0.000, B 0.000, C 0.000 }
gfCNCPoint6[5556] = {X 214.4548, Y 92.8953, Z -8.0000, A 0.000, B 0.000, C 0.000 }
gfCNCPoint6[5557] = {X 215.5118, Y 92.8342, Z -8.0000, A 0.000, B 0.000, C 0.000 }
gfCNCPoint6[5558] = {X 216.2107, Y 92.7578, Z -8.0000, A 0.000, B 0.000, C 0.000 }
gfCNCPoint6[5559] = {X 216.8837, Y 92.5542, Z -8.0000, A 0.000, B 0.000, C 0.000 }
gfCNCPoint6[5560] = {X 217.5076, Y 92.2302, Z -8.0000, A 0.000, B 0.000, C 0.000 }
gfCNCPoint6[5561] = {X 223.0478, Y 88.6549, Z -8.0000, A 0.000, B 0.000, C 0.000 }
gfCNCPoint6[5562] = {X 246.1774, Y 73.8654, Z -8.0000, A 0.000, B 0.000, C 0.000 }
gfCNCPoint6[5563] = {X 221.6900, Y 64.2565, Z -8.0000, A 0.000, B 0.000, C 0.000 }
gfCNCPoint6[5564] = {X 219.9051, Y 63.6593, Z -8.0000, A 0.000, B 0.000, C 0.000 }
gfCNCPoint6[5565] = {X 218.0637, Y 63.2693, Z -8.0000, A 0.000, B 0.000, C 0.000 }
gfCNCPoint6[5566] = {X 216.1900, Y 63.0917, Z -8.0000, A 0.000, B 0.000, C 0.000 }
gfCNCPoint6[5567] = {X 215.2926, Y 62.9624, Z -8.0000, A 0.000, B 0.000, C 0.000 }
gfCNCPoint6[5568] = {X 214.4445, Y 62.6418, Z -8.0000, A 0.000, B 0.000, C 0.000 }
gfCNCPoint6[5569] = {X 213.6860, Y 62.1451, Z -8.0000, A 0.000, B 0.000, C 0.000 }
gfCNCPoint6[5570] = {X 213.0531, Y 61.4958, Z -8.0000, A 0.000, B 0.000, C 0.000 }
gfCNCPoint6[5571] = {X 212.5760, Y 60.7249, Z -8.0000, A 0.000, B 0.000, C 0.000 }
gfCNCPoint6[5572] = {X 212.2772, Y 59.8688, Z -8.0000, A 0.000, B 0.000, C 0.000 }
gfCNCPoint6[5573] = {X 212.1710, Y 58.9684, Z -8.0000, A 0.000, B 0.000, C 0.000 }
gfCNCPoint6[5574] = {X 212.1708, Y 58.0000, Z -8.0000, A 0.000, B 0.000, C 0.000 }
gfCNCPoint6[5575] = {X 212.2751, Y 57.0743, Z -8.0000, A 0.000, B 0.000, C 0.000 }
gfCNCPoint6[5576] = {X 212.5828, Y 56.1950, Z -8.0000, A 0.000, B 0.000, C 0.000 }
gfCNCPoint6[5577] = {X 213.0784, Y 55.4063, Z -8.0000, A 0.000, B 0.000, C 0.000 }
gfCNCPoint6[5578] = {X 213.7371, Y 54.7476, Z -8.0000, A 0.000, B 0.000, C 0.000 }
gfCNCPoint6[5579] = {X 214.5259, Y 54.2520, Z -8.0000, A 0.000, B 0.000, C 0.000 }
gfCNCPoint6[5580] = {X 215.4051, Y 53.9443, Z -8.0000, A 0.000, B 0.000, C 0.000 }
gfCNCPoint6[5581] = {X 216.3308, Y 53.8400, Z -8.0000, A 0.000, B 0.000, C 0.000 }
gfCNCPoint6[5582] = {X 237.2617, Y 53.8400, Z -8.0000, A 0.000, B 0.000, C 0.000 }
gfCNCPoint6[5583] = {X 238.1874, Y 53.9443, Z -8.0000, A 0.000, B 0.000, C 0.000 }
gfCNCPoint6[5584] = {X 239.0666, Y 54.2520, Z -8.0000, A 0.000, B 0.000, C 0.000 }
gfCNCPoint6[5585] = {X 239.8554, Y 54.7476, Z -8.0000, A 0.000, B 0.000, C 0.000 }
gfCNCPoint6[5586] = {X 240.5141, Y 55.4063, Z -8.0000, A 0.000, B 0.000, C 0.000 }
gfCNCPoint6[5587] = {X 241.0097, Y 56.1950, Z -8.0000, A 0.000, B 0.000, C 0.000 }
gfCNCPoint6[5588] = {X 241.3174, Y 57.0743, Z -8.0000, A 0.000, B 0.000, C 0.000 }
gfCNCPoint6[5589] = {X 241.4217, Y 58.0000, Z -8.0000, A 0.000, B 0.000, C 0.000 }
gfCNCPoint6[5590] = {X 241.4217, Y 58.3409, Z -8.0000, A 0.000, B 0.000, C 0.000 }
gfCNCPoint6[5591] = {X 248.0566, Y 60.9282, Z -8.0000, A 0.000, B 0.000, C 0.000 }
gfCNCPoint6[5592] = {X 275.7915, Y 71.9367, Z -8.0000, A 0.000, B 0.000, C 0.000 }
gfCNCPoint6[5593] = {X 275.7933, Y 63.0708, Z -8.0000, A 0.000, B 0.000, C 0.000 }
gfCNCPoint6[5594] = {X 275.6907, Y 63.0586, Z -8.0000, A 0.000, B 0.000, C 0.000 }
gfCNCPoint6[5595] = {X 275.5885, Y 63.0439, Z -8.0000, A 0.000, B 0.000, C 0.000 }
gfCNCPoint6[5596] = {X 274.6511, Y 62.7817, Z -8.0000, A 0.000, B 0.000, C 0.000 }
gfCNCPoint6[5597] = {X 273.8004, Y 62.3089, Z -8.0000, A 0.000, B 0.000, C 0.000 }
gfCNCPoint6[5598] = {X 273.0827, Y 61.6513, Z -8.0000, A 0.000, B 0.000, C 0.000 }
gfCNCPoint6[5599] = {X 272.5376, Y 60.8450, Z -8.0000, A 0.000, B 0.000, C 0.000 }
gfCNCPoint6[5600] = {X 272.1947, Y 59.9341, Z -8.0000, A 0.000, B 0.000, C 0.000 }
gfCNCPoint6[5601] = {X 272.0728, Y 58.9684, Z -8.0000, A 0.000, B 0.000, C 0.000 }
gfCNCPoint6[5602] = {X 272.0727, Y 58.0000, Z -8.0000, A 0.000, B 0.000, C 0.000 }
gfCNCPoint6[5603] = {X 272.1770, Y 57.0743, Z -8.0000, A 0.000, B 0.000, C 0.000 }
gfCNCPoint6[5604] = {X 272.4847, Y 56.1950, Z -8.0000, A 0.000, B 0.000, C 0.000 }
gfCNCPoint6[5605] = {X 272.9803, Y 55.4063, Z -8.0000, A 0.000, B 0.000, C 0.000 }
gfCNCPoint6[5606] = {X 273.6390, Y 54.7476, Z -8.0000, A 0.000, B 0.000, C 0.000 }
gfCNCPoint6[5607] = {X 274.4277, Y 54.2520, Z -8.0000, A 0.000, B 0.000, C 0.000 }
gfCNCPoint6[5608] = {X 275.3070, Y 53.9443, Z -8.0000, A 0.000, B 0.000, C 0.000 }
gfCNCPoint6[5609] = {X 276.2327, Y 53.8400, Z -8.0000, A 0.000, B 0.000, C 0.000 }
gfCNCPoint6[5610] = {X 292.7731, Y 53.8400, Z -8.0000, A 0.000, B 0.000, C 0.000 }
gfCNCPoint6[5611] = {X 293.6988, Y 53.9443, Z -8.0000, A 0.000, B 0.000, C 0.000 }
gfCNCPoint6[5612] = {X 294.5780, Y 54.2520, Z -8.0000, A 0.000, B 0.000, C 0.000 }
gfCNCPoint6[5613] = {X 295.3668, Y 54.7476, Z -8.0000, A 0.000, B 0.000, C 0.000 }
gfCNCPoint6[5614] = {X 296.0255, Y 55.4063, Z -8.0000, A 0.000, B 0.000, C 0.000 }
gfCNCPoint6[5615] = {X 296.5211, Y 56.1950, Z -8.0000, A 0.000, B 0.000, C 0.000 }
gfCNCPoint6[5616] = {X 296.8288, Y 57.0743, Z -8.0000, A 0.000, B 0.000, C 0.000 }
gfCNCPoint6[5617] = {X 296.9331, Y 58.0000, Z -8.0000, A 0.000, B 0.000, C 0.000 }
gfCNCPoint6[5618] = {X 296.9331, Y 58.9345, Z -8.0000, A 0.000, B 0.000, C 0.000 }
gfCNCPoint6[5619] = {X 296.8158, Y 59.9063, Z -8.0000, A 0.000, B 0.000, C 0.000 }
gfCNCPoint6[5620] = {X 296.4755, Y 60.8241, Z -8.0000, A 0.000, B 0.000, C 0.000 }
gfCNCPoint6[5621] = {X 295.9309, Y 61.6375, Z -8.0000, A 0.000, B 0.000, C 0.000 }
gfCNCPoint6[5622] = {X 295.2119, Y 62.3017, Z -8.0000, A 0.000, B 0.000, C 0.000 }
gfCNCPoint6[5623] = {X 294.3580, Y 62.7803, Z -8.0000, A 0.000, B 0.000, C 0.000 }
gfCNCPoint6[5624] = {X 293.4162, Y 63.0471, Z -8.0000, A 0.000, B 0.000, C 0.000 }
gfCNCPoint6[5625] = {X 293.3194, Y 63.0614, Z -8.0000, A 0.000, B 0.000, C 0.000 }
gfCNCPoint6[5626] = {X 293.2223, Y 63.0734, Z -8.0000, A 0.000, B 0.000, C 0.000 }
gfCNCPoint6[5627] = {X 293.2141, Y 63.1614, Z -8.0000, A 0.000, B 0.000, C 0.000 }
gfCNCPoint6[5628] = {X 293.2250, Y 92.9200, Z -8.0000, A 0.000, B 0.000, C 0.000 }
gfCNCPoint6[5629] = {X 293.3204, Y 92.9322, Z -8.0000, A 0.000, B 0.000, C 0.000 }
gfCNCPoint6[5630] = {X 293.4155, Y 92.9465, Z -8.0000, A 0.000, B 0.000, C 0.000 }
gfCNCPoint6[5631] = {X 294.3569, Y 93.2159, Z -8.0000, A 0.000, B 0.000, C 0.000 }
gfCNCPoint6[5632] = {X 295.2102, Y 93.6963, Z -8.0000, A 0.000, B 0.000, C 0.000 }
gfCNCPoint6[5633] = {X 295.9287, Y 94.3616, Z -8.0000, A 0.000, B 0.000, C 0.000 }
gfCNCPoint6[5634] = {X 296.4733, Y 95.1754, Z -8.0000, A 0.000, B 0.000, C 0.000 }
gfCNCPoint6[5635] = {X 296.8143, Y 96.0933, Z -8.0000, A 0.000, B 0.000, C 0.000 }
gfCNCPoint6[5636] = {X 296.9331, Y 97.0653, Z -8.0000, A 0.000, B 0.000, C 0.000 }
gfCNCPoint6[5637] = {X 296.9331, Y 98.0000, Z -8.0000, A 0.000, B 0.000, C 0.000 }
gfCNCPoint6[5638] = {X 296.8288, Y 98.9257, Z -8.0000, A 0.000, B 0.000, C 0.000 }
gfCNCPoint6[5639] = {X 296.5211, Y 99.8050, Z -8.0000, A 0.000, B 0.000, C 0.000 }
gfCNCPoint6[5640] = {X 296.0255, Y 100.5937, Z -8.0000, A 0.000, B 0.000, C 0.000 }
gfCNCPoint6[5641] = {X 295.3668, Y 101.2524, Z -8.0000, A 0.000, B 0.000, C 0.000 }
gfCNCPoint6[5642] = {X 294.5780, Y 101.7480, Z -8.0000, A 0.000, B 0.000, C 0.000 }
gfCNCPoint6[5643] = {X 293.6988, Y 102.0557, Z -8.0000, A 0.000, B 0.000, C 0.000 }
gfCNCPoint6[5644] = {X 292.7731, Y 102.1600, Z -8.0000, A 0.000, B 0.000, C 0.000 }
gfCNCPoint6[5645] = {X 276.2327, Y 102.1600, Z -8.0000, A 0.000, B 0.000, C 0.000 }
gfCNCPoint6[5646] = {X 275.3070, Y 102.0557, Z -8.0000, A 0.000, B 0.000, C 0.000 }
gfCNCPoint6[5647] = {X 274.4277, Y 101.7480, Z -8.0000, A 0.000, B 0.000, C 0.000 }
gfCNCPoint6[5648] = {X 273.6390, Y 101.2524, Z -8.0000, A 0.000, B 0.000, C 0.000 }
gfCNCPoint6[5649] = {X 272.9803, Y 100.5937, Z -8.0000, A 0.000, B 0.000, C 0.000 }
gfCNCPoint6[5650] = {X 272.4847, Y 99.8050, Z -8.0000, A 0.000, B 0.000, C 0.000 }
gfCNCPoint6[5651] = {X 272.1770, Y 98.9257, Z -8.0000, A 0.000, B 0.000, C 0.000 }
gfCNCPoint6[5652] = {X 272.0727, Y 98.0000, Z -8.0000, A 0.000, B 0.000, C 0.000 }
gfCNCPoint6[5653] = {X 272.0727, Y 97.0658, Z -8.0000, A 0.000, B 0.000, C 0.000 }
gfCNCPoint6[5654] = {X 272.1634, Y 96.2021, Z -8.0000, A 0.000, B 0.000, C 0.000 }
gfCNCPoint6[5655] = {X 272.4314, Y 95.3761, Z -8.0000, A 0.000, B 0.000, C 0.000 }
gfCNCPoint6[5656] = {X 272.8651, Y 94.6236, Z -8.0000, A 0.000, B 0.000, C 0.000 }
gfCNCPoint6[5657] = {X 273.4455, Y 93.9777, Z -8.0000, A 0.000, B 0.000, C 0.000 }
gfCNCPoint6[5658] = {X 274.1475, Y 93.4663, Z -8.0000, A 0.000, B 0.000, C 0.000 }
gfCNCPoint6[5659] = {X 274.9403, Y 93.1118, Z -8.0000, A 0.000, B 0.000, C 0.000 }
gfCNCPoint6[5660] = {X 275.7894, Y 92.9296, Z -8.0000, A 0.000, B 0.000, C 0.000 }
gfCNCPoint6[5661] = {X 275.7894, Y 85.4858, Z -8.0000, A 0.000, B 0.000, C 0.000 }
gfCNCPoint6[5662] = {X 262.6239, Y 80.3250, Z -8.0000, A 0.000, B 0.000, C 0.000 }
gfCNCPoint6[5663] = {X 237.6372, Y 96.5017, Z -8.0000, A 0.000, B 0.000, C 0.000 }
gfCNCPoint6[5664] = {X 237.6398, Y 97.0655, Z -8.0000, A 0.000, B 0.000, C 0.000 }
gfCNCPoint6[5665] = {X 237.6398, Y 98.0000, Z -8.0000, A 0.000, B 0.000, C 0.000 }
gfCNCPoint6[5666] = {X 237.5355, Y 98.9257, Z -8.0000, A 0.000, B 0.000, C 0.000 }
gfCNCPoint6[5667] = {X 237.2278, Y 99.8050, Z -8.0000, A 0.000, B 0.000, C 0.000 }
gfCNCPoint6[5668] = {X 236.7322, Y 100.5937, Z -8.0000, A 0.000, B 0.000, C 0.000 }
gfCNCPoint6[5669] = {X 236.0735, Y 101.2524, Z -8.0000, A 0.000, B 0.000, C 0.000 }
gfCNCPoint6[5670] = {X 235.2847, Y 101.7480, Z -8.0000, A 0.000, B 0.000, C 0.000 }
gfCNCPoint6[5671] = {X 234.4055, Y 102.0557, Z -8.0000, A 0.000, B 0.000, C 0.000 }
gfCNCPoint6[5672] = {X 233.4798, Y 102.1600, Z -8.0000, A 0.000, B 0.000, C 0.000 }
gfCNCPoint6[5673] = {X 214.1790, Y 102.1600, Z -8.0000, A 0.000, B 0.000, C 0.000 }
gfCNCPoint6[5674] = {X 213.7860, Y 102.1414, Z -8.0000, A 0.000, B 0.000, C 0.000 }
gfCNCPoint6[5675] = {X 213.3966, Y 102.0857, Z -8.0000, A 0.000, B 0.000, C 0.000 }
gfCNCPoint6[5676] = {X 213.0071, Y 102.1414, Z -8.0000, A 0.000, B 0.000, C 0.000 }
gfCNCPoint6[5677] = {X 212.6141, Y 102.1600, Z -8.0000, A 0.000, B 0.000, C 0.000 }
gfCNCPoint6[5678] = {X 194.9870, Y 102.1600, Z -8.0000, A 0.000, B 0.000, C 0.000 }
gfCNCPoint6[5679] = {X 194.0613, Y 102.0557, Z -8.0000, A 0.000, B 0.000, C 0.000 }
gfCNCPoint6[5680] = {X 193.1820, Y 101.7480, Z -8.0000, A 0.000, B 0.000, C 0.000 }
gfCNCPoint6[5681] = {X 192.3932, Y 101.2524, Z -8.0000, A 0.000, B 0.000, C 0.000 }
gfCNCPoint6[5682] = {X 191.7345, Y 100.5937, Z -8.0000, A 0.000, B 0.000, C 0.000 }
gfCNCPoint6[5683] = {X 191.2389, Y 99.8050, Z -8.0000, A 0.000, B 0.000, C 0.000 }
gfCNCPoint6[5684] = {X 190.9313, Y 98.9257, Z -8.0000, A 0.000, B 0.000, C 0.000 }
gfCNCPoint6[5685] = {X 190.8270, Y 98.0000, Z -8.0000, A 0.000, B 0.000, C 0.000 }
gfCNCPoint6[5686] = {X 190.8270, Y 97.0659, Z -8.0000, A 0.000, B 0.000, C 0.000 }
gfCNCPoint6[5687] = {X 190.9241, Y 96.1723, Z -8.0000, A 0.000, B 0.000, C 0.000 }
gfCNCPoint6[5688] = {X 191.2109, Y 95.3203, Z -8.0000, A 0.000, B 0.000, C 0.000 }
gfCNCPoint6[5689] = {X 191.6741, Y 94.5499, Z -8.0000, A 0.000, B 0.000, C 0.000 }
gfCNCPoint6[5690] = {X 191.7354, Y 94.4712, Z -8.0000, A 0.000, B 0.000, C 0.000 }
gfCNCPoint6[5691] = {X 191.7986, Y 94.3939, Z -8.0000, A 0.000, B 0.000, C 0.000 }
gfCNCPoint6[5692] = {X 188.6351, Y 90.9402, Z -8.0000, A 0.000, B 0.000, C 0.000 }
gfCNCPoint6[5693] = {X 150.0187, Y 90.9402, Z -8.0000, A 0.000, B 0.000, C 0.000 }
gfCNCPoint6[5694] = {X 146.9343, Y 94.3574, Z -8.0000, A 0.000, B 0.000, C 0.000 }
gfCNCPoint6[5695] = {X 147.4808, Y 95.1721, Z -8.0000, A 0.000, B 0.000, C 0.000 }
gfCNCPoint6[5696] = {X 147.8220, Y 96.0918, Z -8.0000, A 0.000, B 0.000, C 0.000 }
gfCNCPoint6[5697] = {X 147.9391, Y 97.0657, Z -8.0000, A 0.000, B 0.000, C 0.000 }
gfCNCPoint6[5698] = {X 147.9391, Y 98.0000, Z -8.0000, A 0.000, B 0.000, C 0.000 }
gfCNCPoint6[5699] = {X 147.8348, Y 98.9257, Z -8.0000, A 0.000, B 0.000, C 0.000 }
gfCNCPoint6[5700] = {X 147.5271, Y 99.8050, Z -8.0000, A 0.000, B 0.000, C 0.000 }
gfCNCPoint6[5701] = {X 147.0315, Y 100.5937, Z -8.0000, A 0.000, B 0.000, C 0.000 }
gfCNCPoint6[5702] = {X 146.3728, Y 101.2524, Z -8.0000, A 0.000, B 0.000, C 0.000 }
gfCNCPoint6[5703] = {X 145.5841, Y 101.7480, Z -8.0000, A 0.000, B 0.000, C 0.000 }
gfCNCPoint6[5704] = {X 144.7048, Y 102.0557, Z -8.0000, A 0.000, B 0.000, C 0.000 }
gfCNCPoint6[5705] = {X 143.7791, Y 102.1600, Z -8.0000, A 0.000, B 0.000, C 0.000 }
gfCNCPoint6[5706] = {X 125.0000, Y 102.1600, Z -8.0000, A 0.000, B 0.000, C 0.000 }
gfCNCPoint6[5707] = {X 124.0743, Y 102.0557, Z -8.0000, A 0.000, B 0.000, C 0.000 }
gfCNCPoint6[5708] = {X 123.1950, Y 101.7480, Z -8.0000, A 0.000, B 0.000, C 0.000 }
gfCNCPoint6[5709] = {X 122.4063, Y 101.2524, Z -8.0000, A 0.000, B 0.000, C 0.000 }
gfCNCPoint6[5710] = {X 121.7476, Y 100.5937, Z -8.0000, A 0.000, B 0.000, C 0.000 }
gfCNCPoint6[5711] = {X 121.2520, Y 99.8050, Z -8.0000, A 0.000, B 0.000, C 0.000 }
gfCNCPoint6[5712] = {X 120.9443, Y 98.9257, Z -8.0000, A 0.000, B 0.000, C 0.000 }
gfCNCPoint6[5713] = {X 120.8400, Y 98.0000, Z -8.0000, A 0.000, B 0.000, C 0.000 }
gfCNCPoint6[5714] = {X 120.8400, Y 97.0659, Z -8.0000, A 0.000, B 0.000, C 0.000 }
gfCNCPoint6[5715] = {X 120.9405, Y 96.1570, Z -8.0000, A 0.000, B 0.000, C 0.000 }
gfCNCPoint6[5716] = {X 121.2372, Y 95.2920, Z -8.0000, A 0.000, B 0.000, C 0.000 }
gfCNCPoint6[5717] = {X 121.7157, Y 94.5127, Z -8.0000, A 0.000, B 0.000, C 0.000 }
gfCNCPoint6[5718] = {X 122.3530, Y 93.8567, Z -8.0000, A 0.000, B 0.000, C 0.000 }
gfCNCPoint6[5719] = {X 123.1181, Y 93.3559, Z -8.0000, A 0.000, B 0.000, C 0.000 }
gfCNCPoint6[5720] = {X 123.9742, Y 93.0344, Z -8.0000, A 0.000, B 0.000, C 0.000 }
gfCNCPoint6[5721] = {X 124.8799, Y 92.9077, Z -8.0000, A 0.000, B 0.000, C 0.000 }
gfCNCPoint6[5722] = {X 124.9137, Y 92.8887, Z -8.0000, A 0.000, B 0.000, C 0.000 }
gfCNCPoint6[5723] = {X 124.9511, Y 92.8784, Z -8.0000, A 0.000, B 0.000, C 0.000 }
gfCNCPoint6[5724] = {X 125.4717, Y 92.8012, Z -8.0000, A 0.000, B 0.000, C 0.000 }
gfCNCPoint6[5725] = {X 126.3311, Y 92.6555, Z -8.0000, A 0.000, B 0.000, C 0.000 }
gfCNCPoint6[5726] = {X 127.1784, Y 92.4508, Z -8.0000, A 0.000, B 0.000, C 0.000 }
gfCNCPoint6[5727] = {X 128.3866, Y 91.3171, Z -8.0000, A 0.000, B 0.000, C 0.000 }
gfCNCPoint6[5728] = {X 129.5302, Y 90.1183, Z -8.0000, A 0.000, B 0.000, C 0.000 }
gfCNCPoint6[5729] = {X 140.7976, Y 77.7459, Z -8.0000, A 0.000, B 0.000, C 0.000 }
gfCNCPoint6[5730] = {X 137.8402, Y 75.0526, Z -8.0000, A 0.000, B 0.000, C 0.000 }
gfCNCPoint6[5731] = {X 140.8568, Y 77.7998, Z -8.0000, A 0.000, B 0.000, C 0.000 }
gfCNCPoint6[5732] = {X 155.9345, Y 61.2435, Z -8.0000, A 0.000, B 0.000, C 0.000 }
gfCNCPoint6[5733] = {X 155.5462, Y 60.5375, Z -8.0000, A 0.000, B 0.000, C 0.000 }
gfCNCPoint6[5734] = {X 155.3043, Y 59.7689, Z -8.0000, A 0.000, B 0.000, C 0.000 }
gfCNCPoint6[5735] = {X 155.2181, Y 58.9678, Z -8.0000, A 0.000, B 0.000, C 0.000 }
gfCNCPoint6[5736] = {X 155.2180, Y 58.0000, Z -8.0000, A 0.000, B 0.000, C 0.000 }
gfCNCPoint6[5737] = {X 155.3203, Y 57.0921, Z -8.0000, A 0.000, B 0.000, C 0.000 }
gfCNCPoint6[5738] = {X 155.6220, Y 56.2298, Z -8.0000, A 0.000, B 0.000, C 0.000 }
gfCNCPoint6[5739] = {X 156.1081, Y 55.4562, Z -8.0000, A 0.000, B 0.000, C 0.000 }
gfCNCPoint6[5740] = {X 156.7541, Y 54.8101, Z -8.0000, A 0.000, B 0.000, C 0.000 }
gfCNCPoint6[5741] = {X 157.5277, Y 54.3240, Z -8.0000, A 0.000, B 0.000, C 0.000 }
gfCNCPoint6[5742] = {X 158.3901, Y 54.0223, Z -8.0000, A 0.000, B 0.000, C 0.000 }
gfCNCPoint6[5743] = {X 159.2980, Y 53.9200, Z -8.0000, A 0.000, B 0.000, C 0.000 }
gfCNCPoint6[5744] = {X 178.5335, Y 53.9200, Z -8.0000, A 0.000, B 0.000, C 0.000 }
gfCNCPoint6[5745] = {X 179.4414, Y 54.0223, Z -8.0000, A 0.000, B 0.000, C 0.000 }
gfCNCPoint6[5746] = {X 180.3037, Y 54.3240, Z -8.0000, A 0.000, B 0.000, C 0.000 }
gfCNCPoint6[5747] = {X 181.0773, Y 54.8101, Z -8.0000, A 0.000, B 0.000, C 0.000 }
gfCNCPoint6[5748] = {X 181.7234, Y 55.4562, Z -8.0000, A 0.000, B 0.000, C 0.000 }
gfCNCPoint6[5749] = {X 182.2095, Y 56.2298, Z -8.0000, A 0.000, B 0.000, C 0.000 }
gfCNCPoint6[5750] = {X 182.5112, Y 57.0921, Z -8.0000, A 0.000, B 0.000, C 0.000 }
gfCNCPoint6[5751] = {X 182.6135, Y 58.0000, Z -8.0000, A 0.000, B 0.000, C 0.000 }
gfCNCPoint6[5752] = {X 182.6135, Y 58.9342, Z -8.0000, A 0.000, B 0.000, C 0.000 }
gfCNCPoint6[5753] = {X 182.5335, Y 59.7380, Z -8.0000, A 0.000, B 0.000, C 0.000 }
gfCNCPoint6[5754] = {X 182.2967, Y 60.5103, Z -8.0000, A 0.000, B 0.000, C 0.000 }
gfCNCPoint6[5755] = {X 181.9125, Y 61.2208, Z -8.0000, A 0.000, B 0.000, C 0.000 }
gfCNCPoint6[5756] = {X 209.1172, Y 90.9189, Z -8.0000, A 0.000, B 0.000, C 0.000 }
gfCNCPoint6[5757] = {X 209.7978, Y 91.6239, Z -8.0000, A 0.000, B 0.000, C 0.000 }
gfCNCPoint6[5758] = {X 210.5143, Y 92.2923, Z -8.0000, A 0.000, B 0.000, C 0.000 }
gfCNCPoint6[5759] = {X 210.9611, Y 92.5947, Z -8.0000, A 0.000, B 0.000, C 0.000 }
gfCNCPoint6[5760] = {X 211.4705, Y 92.7725, Z -8.0000, A 0.000, B 0.000, C 0.000 }
gfCNCPoint6[5761] = {X 212.0678, Y 92.8976, Z -8.0000, A 0.000, B 0.000, C 0.000 }
gfCNCPoint6[5762] = {X 213.3906, Y 93.0642, Z -8.0000, A 0.000, B 0.000, C 0.000 }
gfCNCPoint6[5763] = {X 213.4133, Y 93.0581, Z -8.0000, A 0.000, B 0.000, C 0.000 }
gfCNCPoint6[5764] = {X 214.4631, Y 92.9749, Z -8.0000, A 0.000, B 0.000, C 0.000 }
gfCNCPoint6[5765] = {X 215.5144, Y 92.9142, Z -8.0000, A 0.000, B 0.000, C 0.000 }
gfCNCPoint6[5766] = {X 216.2276, Y 92.8360, Z -8.0000, A 0.000, B 0.000, C 0.000 }
gfCNCPoint6[5767] = {X 216.9143, Y 92.6281, Z -8.0000, A 0.000, B 0.000, C 0.000 }
gfCNCPoint6[5768] = {X 217.5510, Y 92.2975, Z -8.0000, A 0.000, B 0.000, C 0.000 }
gfCNCPoint6[5769] = {X 223.0910, Y 88.7222, Z -8.0000, A 0.000, B 0.000, C 0.000 }
gfCNCPoint6[5770] = {X 246.3527, Y 73.8483, Z -8.0000, A 0.000, B 0.000, C 0.000 }
gfCNCPoint6[5771] = {X 221.7196, Y 64.1822, Z -8.0000, A 0.000, B 0.000, C 0.000 }
gfCNCPoint6[5772] = {X 219.9260, Y 63.5821, Z -8.0000, A 0.000, B 0.000, C 0.000 }
gfCNCPoint6[5773] = {X 218.0758, Y 63.1902, Z -8.0000, A 0.000, B 0.000, C 0.000 }
gfCNCPoint6[5774] = {X 216.1929, Y 63.0117, Z -8.0000, A 0.000, B 0.000, C 0.000 }
gfCNCPoint6[5775] = {X 215.3127, Y 62.8850, Z -8.0000, A 0.000, B 0.000, C 0.000 }
gfCNCPoint6[5776] = {X 214.4809, Y 62.5706, Z -8.0000, A 0.000, B 0.000, C 0.000 }
gfCNCPoint6[5777] = {X 213.7369, Y 62.0834, Z -8.0000, A 0.000, B 0.000, C 0.000 }
gfCNCPoint6[5778] = {X 213.1162, Y 61.4466, Z -8.0000, A 0.000, B 0.000, C 0.000 }
gfCNCPoint6[5779] = {X 212.6482, Y 60.6905, Z -8.0000, A 0.000, B 0.000, C 0.000 }
gfCNCPoint6[5780] = {X 212.3552, Y 59.8509, Z -8.0000, A 0.000, B 0.000, C 0.000 }
gfCNCPoint6[5781] = {X 212.2509, Y 58.9678, Z -8.0000, A 0.000, B 0.000, C 0.000 }
gfCNCPoint6[5782] = {X 212.2508, Y 58.0000, Z -8.0000, A 0.000, B 0.000, C 0.000 }
gfCNCPoint6[5783] = {X 212.3531, Y 57.0921, Z -8.0000, A 0.000, B 0.000, C 0.000 }
gfCNCPoint6[5784] = {X 212.6549, Y 56.2298, Z -8.0000, A 0.000, B 0.000, C 0.000 }
gfCNCPoint6[5785] = {X 213.1409, Y 55.4562, Z -8.0000, A 0.000, B 0.000, C 0.000 }
gfCNCPoint6[5786] = {X 213.7870, Y 54.8101, Z -8.0000, A 0.000, B 0.000, C 0.000 }
gfCNCPoint6[5787] = {X 214.5606, Y 54.3240, Z -8.0000, A 0.000, B 0.000, C 0.000 }
gfCNCPoint6[5788] = {X 215.4229, Y 54.0223, Z -8.0000, A 0.000, B 0.000, C 0.000 }
gfCNCPoint6[5789] = {X 216.3308, Y 53.9200, Z -8.0000, A 0.000, B 0.000, C 0.000 }
gfCNCPoint6[5790] = {X 237.2617, Y 53.9200, Z -8.0000, A 0.000, B 0.000, C 0.000 }
gfCNCPoint6[5791] = {X 238.1696, Y 54.0223, Z -8.0000, A 0.000, B 0.000, C 0.000 }
gfCNCPoint6[5792] = {X 239.0319, Y 54.3240, Z -8.0000, A 0.000, B 0.000, C 0.000 }
gfCNCPoint6[5793] = {X 239.8055, Y 54.8101, Z -8.0000, A 0.000, B 0.000, C 0.000 }
gfCNCPoint6[5794] = {X 240.4516, Y 55.4562, Z -8.0000, A 0.000, B 0.000, C 0.000 }
gfCNCPoint6[5795] = {X 240.9376, Y 56.2298, Z -8.0000, A 0.000, B 0.000, C 0.000 }
gfCNCPoint6[5796] = {X 241.2394, Y 57.0921, Z -8.0000, A 0.000, B 0.000, C 0.000 }
gfCNCPoint6[5797] = {X 241.3417, Y 58.0000, Z -8.0000, A 0.000, B 0.000, C 0.000 }
gfCNCPoint6[5798] = {X 241.3417, Y 58.3956, Z -8.0000, A 0.000, B 0.000, C 0.000 }
gfCNCPoint6[5799] = {X 248.0273, Y 61.0026, Z -8.0000, A 0.000, B 0.000, C 0.000 }
gfCNCPoint6[5800] = {X 275.8715, Y 72.0545, Z -8.0000, A 0.000, B 0.000, C 0.000 }
gfCNCPoint6[5801] = {X 275.8733, Y 62.9982, Z -8.0000, A 0.000, B 0.000, C 0.000 }
gfCNCPoint6[5802] = {X 275.7368, Y 62.9838, Z -8.0000, A 0.000, B 0.000, C 0.000 }
gfCNCPoint6[5803] = {X 275.6009, Y 62.9648, Z -8.0000, A 0.000, B 0.000, C 0.000 }
gfCNCPoint6[5804] = {X 274.6815, Y 62.7077, Z -8.0000, A 0.000, B 0.000, C 0.000 }
gfCNCPoint6[5805] = {X 273.8471, Y 62.2440, Z -8.0000, A 0.000, B 0.000, C 0.000 }
gfCNCPoint6[5806] = {X 273.1433, Y 61.5991, Z -8.0000, A 0.000, B 0.000, C 0.000 }
gfCNCPoint6[5807] = {X 272.6086, Y 60.8083, Z -8.0000, A 0.000, B 0.000, C 0.000 }
gfCNCPoint6[5808] = {X 272.2723, Y 59.9149, Z -8.0000, A 0.000, B 0.000, C 0.000 }
gfCNCPoint6[5809] = {X 272.1528, Y 58.9678, Z -8.0000, A 0.000, B 0.000, C 0.000 }
gfCNCPoint6[5810] = {X 272.1527, Y 58.0000, Z -8.0000, A 0.000, B 0.000, C 0.000 }
gfCNCPoint6[5811] = {X 272.2550, Y 57.0921, Z -8.0000, A 0.000, B 0.000, C 0.000 }
gfCNCPoint6[5812] = {X 272.5567, Y 56.2298, Z -8.0000, A 0.000, B 0.000, C 0.000 }
gfCNCPoint6[5813] = {X 273.0428, Y 55.4562, Z -8.0000, A 0.000, B 0.000, C 0.000 }
gfCNCPoint6[5814] = {X 273.6889, Y 54.8101, Z -8.0000, A 0.000, B 0.000, C 0.000 }
gfCNCPoint6[5815] = {X 274.4624, Y 54.3240, Z -8.0000, A 0.000, B 0.000, C 0.000 }
gfCNCPoint6[5816] = {X 275.3248, Y 54.0223, Z -8.0000, A 0.000, B 0.000, C 0.000 }
gfCNCPoint6[5817] = {X 276.2327, Y 53.9200, Z -8.0000, A 0.000, B 0.000, C 0.000 }
gfCNCPoint6[5818] = {X 292.7731, Y 53.9200, Z -8.0000, A 0.000, B 0.000, C 0.000 }
gfCNCPoint6[5819] = {X 293.6810, Y 54.0223, Z -8.0000, A 0.000, B 0.000, C 0.000 }
gfCNCPoint6[5820] = {X 294.5433, Y 54.3240, Z -8.0000, A 0.000, B 0.000, C 0.000 }
gfCNCPoint6[5821] = {X 295.3169, Y 54.8101, Z -8.0000, A 0.000, B 0.000, C 0.000 }
gfCNCPoint6[5822] = {X 295.9630, Y 55.4562, Z -8.0000, A 0.000, B 0.000, C 0.000 }
gfCNCPoint6[5823] = {X 296.4490, Y 56.2298, Z -8.0000, A 0.000, B 0.000, C 0.000 }
gfCNCPoint6[5824] = {X 296.7508, Y 57.0921, Z -8.0000, A 0.000, B 0.000, C 0.000 }
gfCNCPoint6[5825] = {X 296.8531, Y 58.0000, Z -8.0000, A 0.000, B 0.000, C 0.000 }
gfCNCPoint6[5826] = {X 296.8531, Y 58.9343, Z -8.0000, A 0.000, B 0.000, C 0.000 }
gfCNCPoint6[5827] = {X 296.7380, Y 59.8875, Z -8.0000, A 0.000, B 0.000, C 0.000 }
gfCNCPoint6[5828] = {X 296.4043, Y 60.7877, Z -8.0000, A 0.000, B 0.000, C 0.000 }
gfCNCPoint6[5829] = {X 295.8701, Y 61.5855, Z -8.0000, A 0.000, B 0.000, C 0.000 }
gfCNCPoint6[5830] = {X 295.1649, Y 62.2370, Z -8.0000, A 0.000, B 0.000, C 0.000 }
gfCNCPoint6[5831] = {X 294.3274, Y 62.7065, Z -8.0000, A 0.000, B 0.000, C 0.000 }
gfCNCPoint6[5832] = {X 293.4036, Y 62.9681, Z -8.0000, A 0.000, B 0.000, C 0.000 }
gfCNCPoint6[5833] = {X 293.2764, Y 62.9863, Z -8.0000, A 0.000, B 0.000, C 0.000 }
gfCNCPoint6[5834] = {X 293.1487, Y 63.0006, Z -8.0000, A 0.000, B 0.000, C 0.000 }
gfCNCPoint6[5835] = {X 293.1341, Y 63.1577, Z -8.0000, A 0.000, B 0.000, C 0.000 }
gfCNCPoint6[5836] = {X 293.1451, Y 92.9918, Z -8.0000, A 0.000, B 0.000, C 0.000 }
gfCNCPoint6[5837] = {X 293.2741, Y 93.0066, Z -8.0000, A 0.000, B 0.000, C 0.000 }
gfCNCPoint6[5838] = {X 293.4026, Y 93.0255, Z -8.0000, A 0.000, B 0.000, C 0.000 }
gfCNCPoint6[5839] = {X 294.3261, Y 93.2897, Z -8.0000, A 0.000, B 0.000, C 0.000 }
gfCNCPoint6[5840] = {X 295.1631, Y 93.7610, Z -8.0000, A 0.000, B 0.000, C 0.000 }
gfCNCPoint6[5841] = {X 295.8679, Y 94.4135, Z -8.0000, A 0.000, B 0.000, C 0.000 }
gfCNCPoint6[5842] = {X 296.4021, Y 95.2118, Z -8.0000, A 0.000, B 0.000, C 0.000 }
gfCNCPoint6[5843] = {X 296.7366, Y 96.1122, Z -8.0000, A 0.000, B 0.000, C 0.000 }
gfCNCPoint6[5844] = {X 296.8531, Y 97.0656, Z -8.0000, A 0.000, B 0.000, C 0.000 }
gfCNCPoint6[5845] = {X 296.8531, Y 98.0000, Z -8.0000, A 0.000, B 0.000, C 0.000 }
gfCNCPoint6[5846] = {X 296.7508, Y 98.9079, Z -8.0000, A 0.000, B 0.000, C 0.000 }
gfCNCPoint6[5847] = {X 296.4490, Y 99.7702, Z -8.0000, A 0.000, B 0.000, C 0.000 }
gfCNCPoint6[5848] = {X 295.9630, Y 100.5438, Z -8.0000, A 0.000, B 0.000, C 0.000 }
gfCNCPoint6[5849] = {X 295.3169, Y 101.1899, Z -8.0000, A 0.000, B 0.000, C 0.000 }
gfCNCPoint6[5850] = {X 294.5433, Y 101.6760, Z -8.0000, A 0.000, B 0.000, C 0.000 }
gfCNCPoint6[5851] = {X 293.6810, Y 101.9777, Z -8.0000, A 0.000, B 0.000, C 0.000 }
gfCNCPoint6[5852] = {X 292.7731, Y 102.0800, Z -8.0000, A 0.000, B 0.000, C 0.000 }
gfCNCPoint6[5853] = {X 276.2327, Y 102.0800, Z -8.0000, A 0.000, B 0.000, C 0.000 }
gfCNCPoint6[5854] = {X 275.3248, Y 101.9777, Z -8.0000, A 0.000, B 0.000, C 0.000 }
gfCNCPoint6[5855] = {X 274.4624, Y 101.6760, Z -8.0000, A 0.000, B 0.000, C 0.000 }
gfCNCPoint6[5856] = {X 273.6889, Y 101.1899, Z -8.0000, A 0.000, B 0.000, C 0.000 }
gfCNCPoint6[5857] = {X 273.0428, Y 100.5438, Z -8.0000, A 0.000, B 0.000, C 0.000 }
gfCNCPoint6[5858] = {X 272.5567, Y 99.7702, Z -8.0000, A 0.000, B 0.000, C 0.000 }
gfCNCPoint6[5859] = {X 272.2550, Y 98.9079, Z -8.0000, A 0.000, B 0.000, C 0.000 }
gfCNCPoint6[5860] = {X 272.1527, Y 98.0000, Z -8.0000, A 0.000, B 0.000, C 0.000 }
gfCNCPoint6[5861] = {X 272.1527, Y 97.0658, Z -8.0000, A 0.000, B 0.000, C 0.000 }
gfCNCPoint6[5862] = {X 272.2438, Y 96.2087, Z -8.0000, A 0.000, B 0.000, C 0.000 }
gfCNCPoint6[5863] = {X 272.5129, Y 95.3898, Z -8.0000, A 0.000, B 0.000, C 0.000 }
gfCNCPoint6[5864] = {X 272.9480, Y 94.6458, Z -8.0000, A 0.000, B 0.000, C 0.000 }
gfCNCPoint6[5865] = {X 273.5297, Y 94.0097, Z -8.0000, A 0.000, B 0.000, C 0.000 }
gfCNCPoint6[5866] = {X 274.2321, Y 93.5101, Z -8.0000, A 0.000, B 0.000, C 0.000 }
gfCNCPoint6[5867] = {X 275.0238, Y 93.1692, Z -8.0000, A 0.000, B 0.000, C 0.000 }
gfCNCPoint6[5868] = {X 275.8694, Y 93.0021, Z -8.0000, A 0.000, B 0.000, C 0.000 }
gfCNCPoint6[5869] = {X 275.8694, Y 85.4313, Z -8.0000, A 0.000, B 0.000, C 0.000 }
gfCNCPoint6[5870] = {X 262.6149, Y 80.2355, Z -8.0000, A 0.000, B 0.000, C 0.000 }
gfCNCPoint6[5871] = {X 237.5570, Y 96.4583, Z -8.0000, A 0.000, B 0.000, C 0.000 }
gfCNCPoint6[5872] = {X 237.5598, Y 97.0657, Z -8.0000, A 0.000, B 0.000, C 0.000 }
gfCNCPoint6[5873] = {X 237.5598, Y 98.0000, Z -8.0000, A 0.000, B 0.000, C 0.000 }
gfCNCPoint6[5874] = {X 237.4575, Y 98.9079, Z -8.0000, A 0.000, B 0.000, C 0.000 }
gfCNCPoint6[5875] = {X 237.1557, Y 99.7702, Z -8.0000, A 0.000, B 0.000, C 0.000 }
gfCNCPoint6[5876] = {X 236.6697, Y 100.5438, Z -8.0000, A 0.000, B 0.000, C 0.000 }
gfCNCPoint6[5877] = {X 236.0236, Y 101.1899, Z -8.0000, A 0.000, B 0.000, C 0.000 }
gfCNCPoint6[5878] = {X 235.2500, Y 101.6760, Z -8.0000, A 0.000, B 0.000, C 0.000 }
gfCNCPoint6[5879] = {X 234.3877, Y 101.9777, Z -8.0000, A 0.000, B 0.000, C 0.000 }
gfCNCPoint6[5880] = {X 233.4798, Y 102.0800, Z -8.0000, A 0.000, B 0.000, C 0.000 }
gfCNCPoint6[5881] = {X 214.1790, Y 102.0800, Z -8.0000, A 0.000, B 0.000, C 0.000 }
gfCNCPoint6[5882] = {X 213.7860, Y 102.0610, Z -8.0000, A 0.000, B 0.000, C 0.000 }
gfCNCPoint6[5883] = {X 213.3966, Y 102.0043, Z -8.0000, A 0.000, B 0.000, C 0.000 }
gfCNCPoint6[5884] = {X 213.0072, Y 102.0610, Z -8.0000, A 0.000, B 0.000, C 0.000 }
gfCNCPoint6[5885] = {X 212.6141, Y 102.0800, Z -8.0000, A 0.000, B 0.000, C 0.000 }
gfCNCPoint6[5886] = {X 194.9870, Y 102.0800, Z -8.0000, A 0.000, B 0.000, C 0.000 }
gfCNCPoint6[5887] = {X 194.0791, Y 101.9777, Z -8.0000, A 0.000, B 0.000, C 0.000 }
gfCNCPoint6[5888] = {X 193.2167, Y 101.6760, Z -8.0000, A 0.000, B 0.000, C 0.000 }
gfCNCPoint6[5889] = {X 192.4431, Y 101.1899, Z -8.0000, A 0.000, B 0.000, C 0.000 }
gfCNCPoint6[5890] = {X 191.7971, Y 100.5438, Z -8.0000, A 0.000, B 0.000, C 0.000 }
gfCNCPoint6[5891] = {X 191.3110, Y 99.7702, Z -8.0000, A 0.000, B 0.000, C 0.000 }
gfCNCPoint6[5892] = {X 191.0093, Y 98.9079, Z -8.0000, A 0.000, B 0.000, C 0.000 }
gfCNCPoint6[5893] = {X 190.9070, Y 98.0000, Z -8.0000, A 0.000, B 0.000, C 0.000 }
gfCNCPoint6[5894] = {X 190.9070, Y 97.0659, Z -8.0000, A 0.000, B 0.000, C 0.000 }
gfCNCPoint6[5895] = {X 191.0022, Y 96.1894, Z -8.0000, A 0.000, B 0.000, C 0.000 }
gfCNCPoint6[5896] = {X 191.2835, Y 95.3539, Z -8.0000, A 0.000, B 0.000, C 0.000 }
gfCNCPoint6[5897] = {X 191.7378, Y 94.5983, Z -8.0000, A 0.000, B 0.000, C 0.000 }
gfCNCPoint6[5898] = {X 191.8199, Y 94.4938, Z -8.0000, A 0.000, B 0.000, C 0.000 }
gfCNCPoint6[5899] = {X 191.9053, Y 94.3920, Z -8.0000, A 0.000, B 0.000, C 0.000 }
gfCNCPoint6[5900] = {X 188.6703, Y 90.8602, Z -8.0000, A 0.000, B 0.000, C 0.000 }
gfCNCPoint6[5901] = {X 149.9831, Y 90.8602, Z -8.0000, A 0.000, B 0.000, C 0.000 }
gfCNCPoint6[5902] = {X 146.8273, Y 94.3565, Z -8.0000, A 0.000, B 0.000, C 0.000 }
gfCNCPoint6[5903] = {X 147.3880, Y 95.1669, Z -8.0000, A 0.000, B 0.000, C 0.000 }
gfCNCPoint6[5904] = {X 147.7387, Y 96.0878, Z -8.0000, A 0.000, B 0.000, C 0.000 }
gfCNCPoint6[5905] = {X 147.8591, Y 97.0659, Z -8.0000, A 0.000, B 0.000, C 0.000 }
gfCNCPoint6[5906] = {X 147.8591, Y 98.0000, Z -8.0000, A 0.000, B 0.000, C 0.000 }
gfCNCPoint6[5907] = {X 147.7568, Y 98.9079, Z -8.0000, A 0.000, B 0.000, C 0.000 }
gfCNCPoint6[5908] = {X 147.4551, Y 99.7702, Z -8.0000, A 0.000, B 0.000, C 0.000 }
gfCNCPoint6[5909] = {X 146.9690, Y 100.5438, Z -8.0000, A 0.000, B 0.000, C 0.000 }
gfCNCPoint6[5910] = {X 146.3229, Y 101.1899, Z -8.0000, A 0.000, B 0.000, C 0.000 }
gfCNCPoint6[5911] = {X 145.5494, Y 101.6760, Z -8.0000, A 0.000, B 0.000, C 0.000 }
gfCNCPoint6[5912] = {X 144.6870, Y 101.9777, Z -8.0000, A 0.000, B 0.000, C 0.000 }
gfCNCPoint6[5913] = {X 143.7791, Y 102.0800, Z -8.0000, A 0.000, B 0.000, C 0.000 }
gfCNCPoint6[5914] = {X 125.0000, Y 102.0800, Z -8.0000, A 0.000, B 0.000, C 0.000 }
gfCNCPoint6[5915] = {X 124.0921, Y 101.9777, Z -8.0000, A 0.000, B 0.000, C 0.000 }
gfCNCPoint6[5916] = {X 123.2298, Y 101.6760, Z -8.0000, A 0.000, B 0.000, C 0.000 }
gfCNCPoint6[5917] = {X 122.4562, Y 101.1899, Z -8.0000, A 0.000, B 0.000, C 0.000 }
gfCNCPoint6[5918] = {X 121.8101, Y 100.5438, Z -8.0000, A 0.000, B 0.000, C 0.000 }
gfCNCPoint6[5919] = {X 121.3240, Y 99.7702, Z -8.0000, A 0.000, B 0.000, C 0.000 }
gfCNCPoint6[5920] = {X 121.0223, Y 98.9079, Z -8.0000, A 0.000, B 0.000, C 0.000 }
gfCNCPoint6[5921] = {X 120.9200, Y 98.0000, Z -8.0000, A 0.000, B 0.000, C 0.000 }
gfCNCPoint6[5922] = {X 120.9200, Y 97.0659, Z -8.0000, A 0.000, B 0.000, C 0.000 }
gfCNCPoint6[5923] = {X 121.0193, Y 96.1711, Z -8.0000, A 0.000, B 0.000, C 0.000 }
gfCNCPoint6[5924] = {X 121.3125, Y 95.3199, Z -8.0000, A 0.000, B 0.000, C 0.000 }
gfCNCPoint6[5925] = {X 121.7852, Y 94.5537, Z -8.0000, A 0.000, B 0.000, C 0.000 }
gfCNCPoint6[5926] = {X 122.4144, Y 93.9098, Z -8.0000, A 0.000, B 0.000, C 0.000 }
gfCNCPoint6[5927] = {X 123.1696, Y 93.4196, Z -8.0000, A 0.000, B 0.000, C 0.000 }
gfCNCPoint6[5928] = {X 124.0138, Y 93.1069, Z -8.0000, A 0.000, B 0.000, C 0.000 }
gfCNCPoint6[5929] = {X 124.9061, Y 92.9870, Z -8.0000, A 0.000, B 0.000, C 0.000 }
gfCNCPoint6[5930] = {X 124.9287, Y 92.9712, Z -8.0000, A 0.000, B 0.000, C 0.000 }
gfCNCPoint6[5931] = {X 124.9629, Y 92.9575, Z -8.0000, A 0.000, B 0.000, C 0.000 }
gfCNCPoint6[5932] = {X 125.4828, Y 92.8804, Z -8.0000, A 0.000, B 0.000, C 0.000 }
gfCNCPoint6[5933] = {X 126.3565, Y 92.7319, Z -8.0000, A 0.000, B 0.000, C 0.000 }
gfCNCPoint6[5934] = {X 127.2177, Y 92.5228, Z -8.0000, A 0.000, B 0.000, C 0.000 }
gfCNCPoint6[5935] = {X 128.4363, Y 91.3804, Z -8.0000, A 0.000, B 0.000, C 0.000 }
gfCNCPoint6[5936] = {X 129.5896, Y 90.1719, Z -8.0000, A 0.000, B 0.000, C 0.000 }
gfCNCPoint6[5937] = {X 140.8568, Y 77.7998, Z -8.0000, A 0.000, B 0.000, C 0.000 }
gfCNCPoint6[5938] = {X 137.8994, Y 75.1065, Z -8.0000, A 0.000, B 0.000, C 0.000 }
gfCNCPoint6[5939] = {X 140.9159, Y 77.8537, Z -8.0000, A 0.000, B 0.000, C 0.000 }
gfCNCPoint6[5940] = {X 156.0367, Y 61.2501, Z -8.0000, A 0.000, B 0.000, C 0.000 }
gfCNCPoint6[5941] = {X 155.6321, Y 60.5346, Z -8.0000, A 0.000, B 0.000, C 0.000 }
gfCNCPoint6[5942] = {X 155.3824, Y 59.7516, Z -8.0000, A 0.000, B 0.000, C 0.000 }
gfCNCPoint6[5943] = {X 155.2980, Y 58.9341, Z -8.0000, A 0.000, B 0.000, C 0.000 }
gfCNCPoint6[5944] = {X 155.2980, Y 58.0000, Z -8.0000, A 0.000, B 0.000, C 0.000 }
gfCNCPoint6[5945] = {X 155.3982, Y 57.1099, Z -8.0000, A 0.000, B 0.000, C 0.000 }
gfCNCPoint6[5946] = {X 155.6941, Y 56.2645, Z -8.0000, A 0.000, B 0.000, C 0.000 }
gfCNCPoint6[5947] = {X 156.1706, Y 55.5060, Z -8.0000, A 0.000, B 0.000, C 0.000 }
gfCNCPoint6[5948] = {X 156.8040, Y 54.8727, Z -8.0000, A 0.000, B 0.000, C 0.000 }
gfCNCPoint6[5949] = {X 157.5624, Y 54.3961, Z -8.0000, A 0.000, B 0.000, C 0.000 }
gfCNCPoint6[5950] = {X 158.4079, Y 54.1003, Z -8.0000, A 0.000, B 0.000, C 0.000 }
gfCNCPoint6[5951] = {X 159.2980, Y 54.0000, Z -8.0000, A 0.000, B 0.000, C 0.000 }
gfCNCPoint6[5952] = {X 178.5335, Y 54.0000, Z -8.0000, A 0.000, B 0.000, C 0.000 }
gfCNCPoint6[5953] = {X 179.4236, Y 54.1003, Z -8.0000, A 0.000, B 0.000, C 0.000 }
gfCNCPoint6[5954] = {X 180.2690, Y 54.3961, Z -8.0000, A 0.000, B 0.000, C 0.000 }
gfCNCPoint6[5955] = {X 181.0275, Y 54.8727, Z -8.0000, A 0.000, B 0.000, C 0.000 }
gfCNCPoint6[5956] = {X 181.6608, Y 55.5060, Z -8.0000, A 0.000, B 0.000, C 0.000 }
gfCNCPoint6[5957] = {X 182.1374, Y 56.2645, Z -8.0000, A 0.000, B 0.000, C 0.000 }
gfCNCPoint6[5958] = {X 182.4332, Y 57.1099, Z -8.0000, A 0.000, B 0.000, C 0.000 }
gfCNCPoint6[5959] = {X 182.5335, Y 58.0000, Z -8.0000, A 0.000, B 0.000, C 0.000 }
gfCNCPoint6[5960] = {X 182.5334, Y 58.9671, Z -8.0000, A 0.000, B 0.000, C 0.000 }
gfCNCPoint6[5961] = {X 182.4464, Y 59.7643, Z -8.0000, A 0.000, B 0.000, C 0.000 }
gfCNCPoint6[5962] = {X 182.2022, Y 60.5281, Z -8.0000, A 0.000, B 0.000, C 0.000 }
gfCNCPoint6[5963] = {X 181.8105, Y 61.2279, Z -8.0000, A 0.000, B 0.000, C 0.000 }
gfCNCPoint6[5964] = {X 209.0582, Y 90.9730, Z -8.0000, A 0.000, B 0.000, C 0.000 }
gfCNCPoint6[5965] = {X 209.7417, Y 91.6810, Z -8.0000, A 0.000, B 0.000, C 0.000 }
gfCNCPoint6[5966] = {X 210.4613, Y 92.3522, Z -8.0000, A 0.000, B 0.000, C 0.000 }
gfCNCPoint6[5967] = {X 210.9252, Y 92.6662, Z -8.0000, A 0.000, B 0.000, C 0.000 }
gfCNCPoint6[5968] = {X 211.4541, Y 92.8508, Z -8.0000, A 0.000, B 0.000, C 0.000 }
gfCNCPoint6[5969] = {X 212.0545, Y 92.9765, Z -8.0000, A 0.000, B 0.000, C 0.000 }
gfCNCPoint6[5970] = {X 213.3962, Y 93.1455, Z -8.0000, A 0.000, B 0.000, C 0.000 }
gfCNCPoint6[5971] = {X 213.4273, Y 93.1372, Z -8.0000, A 0.000, B 0.000, C 0.000 }
gfCNCPoint6[5972] = {X 214.4714, Y 93.0545, Z -8.0000, A 0.000, B 0.000, C 0.000 }
gfCNCPoint6[5973] = {X 215.5170, Y 92.9941, Z -8.0000, A 0.000, B 0.000, C 0.000 }
gfCNCPoint6[5974] = {X 216.2445, Y 92.9142, Z -8.0000, A 0.000, B 0.000, C 0.000 }
gfCNCPoint6[5975] = {X 216.9449, Y 92.7020, Z -8.0000, A 0.000, B 0.000, C 0.000 }
gfCNCPoint6[5976] = {X 217.5944, Y 92.3647, Z -8.0000, A 0.000, B 0.000, C 0.000 }
gfCNCPoint6[5977] = {X 223.1343, Y 88.7895, Z -8.0000, A 0.000, B 0.000, C 0.000 }
gfCNCPoint6[5978] = {X 246.5280, Y 73.8311, Z -8.0000, A 0.000, B 0.000, C 0.000 }
gfCNCPoint6[5979] = {X 221.7493, Y 64.1079, Z -8.0000, A 0.000, B 0.000, C 0.000 }
gfCNCPoint6[5980] = {X 219.9471, Y 63.5049, Z -8.0000, A 0.000, B 0.000, C 0.000 }
gfCNCPoint6[5981] = {X 218.0878, Y 63.1111, Z -8.0000, A 0.000, B 0.000, C 0.000 }
gfCNCPoint6[5982] = {X 216.1958, Y 62.9318, Z -8.0000, A 0.000, B 0.000, C 0.000 }
gfCNCPoint6[5983] = {X 215.3283, Y 62.8064, Z -8.0000, A 0.000, B 0.000, C 0.000 }
gfCNCPoint6[5984] = {X 214.5089, Y 62.4951, Z -8.0000, A 0.000, B 0.000, C 0.000 }
gfCNCPoint6[5985] = {X 213.7770, Y 62.0127, Z -8.0000, A 0.000, B 0.000, C 0.000 }
gfCNCPoint6[5986] = {X 213.1677, Y 61.3825, Z -8.0000, A 0.000, B 0.000, C 0.000 }
gfCNCPoint6[5987] = {X 212.7104, Y 60.6348, Z -8.0000, A 0.000, B 0.000, C 0.000 }
gfCNCPoint6[5988] = {X 212.4268, Y 59.8053, Z -8.0000, A 0.000, B 0.000, C 0.000 }
gfCNCPoint6[5989] = {X 212.3308, Y 58.9341, Z -8.0000, A 0.000, B 0.000, C 0.000 }
gfCNCPoint6[5990] = {X 212.3308, Y 58.0000, Z -8.0000, A 0.000, B 0.000, C 0.000 }
gfCNCPoint6[5991] = {X 212.4311, Y 57.1099, Z -8.0000, A 0.000, B 0.000, C 0.000 }
gfCNCPoint6[5992] = {X 212.7269, Y 56.2645, Z -8.0000, A 0.000, B 0.000, C 0.000 }
gfCNCPoint6[5993] = {X 213.2035, Y 55.5060, Z -8.0000, A 0.000, B 0.000, C 0.000 }
gfCNCPoint6[5994] = {X 213.8368, Y 54.8727, Z -8.0000, A 0.000, B 0.000, C 0.000 }
gfCNCPoint6[5995] = {X 214.5953, Y 54.3961, Z -8.0000, A 0.000, B 0.000, C 0.000 }
gfCNCPoint6[5996] = {X 215.4407, Y 54.1003, Z -8.0000, A 0.000, B 0.000, C 0.000 }
gfCNCPoint6[5997] = {X 216.3308, Y 54.0000, Z -8.0000, A 0.000, B 0.000, C 0.000 }
gfCNCPoint6[5998] = {X 237.2617, Y 54.0000, Z -8.0000, A 0.000, B 0.000, C 0.000 }
gfCNCPoint6[5999] = {X 238.1518, Y 54.1003, Z -8.0000, A 0.000, B 0.000, C 0.000 }
gfCNCPoint6[6000] = {X 238.9972, Y 54.3961, Z -8.0000, A 0.000, B 0.000, C 0.000 }
gfCNCPoint6[6001] = {X 239.7556, Y 54.8727, Z -8.0000, A 0.000, B 0.000, C 0.000 }
gfCNCPoint6[6002] = {X 240.3890, Y 55.5060, Z -8.0000, A 0.000, B 0.000, C 0.000 }
gfCNCPoint6[6003] = {X 240.8656, Y 56.2645, Z -8.0000, A 0.000, B 0.000, C 0.000 }
gfCNCPoint6[6004] = {X 241.1614, Y 57.1099, Z -8.0000, A 0.000, B 0.000, C 0.000 }
gfCNCPoint6[6005] = {X 241.2617, Y 58.0000, Z -8.0000, A 0.000, B 0.000, C 0.000 }
gfCNCPoint6[6006] = {X 241.2617, Y 58.4502, Z -8.0000, A 0.000, B 0.000, C 0.000 }
gfCNCPoint6[6007] = {X 247.9980, Y 61.0771, Z -8.0000, A 0.000, B 0.000, C 0.000 }
gfCNCPoint6[6008] = {X 275.9515, Y 72.1724, Z -8.0000, A 0.000, B 0.000, C 0.000 }
gfCNCPoint6[6009] = {X 275.9513, Y 63.0396, Z -8.0000, A 0.000, B 0.000, C 0.000 }
gfCNCPoint6[6010] = {X 275.9573, Y 62.9246, Z -8.0000, A 0.000, B 0.000, C 0.000 }
gfCNCPoint6[6011] = {X 275.7849, Y 62.9089, Z -8.0000, A 0.000, B 0.000, C 0.000 }
gfCNCPoint6[6012] = {X 275.6132, Y 62.8858, Z -8.0000, A 0.000, B 0.000, C 0.000 }
gfCNCPoint6[6013] = {X 274.7069, Y 62.6316, Z -8.0000, A 0.000, B 0.000, C 0.000 }
gfCNCPoint6[6014] = {X 273.8850, Y 62.1726, Z -8.0000, A 0.000, B 0.000, C 0.000 }
gfCNCPoint6[6015] = {X 273.1931, Y 61.5343, Z -8.0000, A 0.000, B 0.000, C 0.000 }
gfCNCPoint6[6016] = {X 272.6696, Y 60.7519, Z -8.0000, A 0.000, B 0.000, C 0.000 }
gfCNCPoint6[6017] = {X 272.3435, Y 59.8689, Z -8.0000, A 0.000, B 0.000, C 0.000 }
gfCNCPoint6[6018] = {X 272.2327, Y 58.9341, Z -8.0000, A 0.000, B 0.000, C 0.000 }
gfCNCPoint6[6019] = {X 272.2327, Y 58.0000, Z -8.0000, A 0.000, B 0.000, C 0.000 }
gfCNCPoint6[6020] = {X 272.3330, Y 57.1099, Z -8.0000, A 0.000, B 0.000, C 0.000 }
gfCNCPoint6[6021] = {X 272.6288, Y 56.2645, Z -8.0000, A 0.000, B 0.000, C 0.000 }
gfCNCPoint6[6022] = {X 273.1054, Y 55.5060, Z -8.0000, A 0.000, B 0.000, C 0.000 }
gfCNCPoint6[6023] = {X 273.7387, Y 54.8727, Z -8.0000, A 0.000, B 0.000, C 0.000 }
gfCNCPoint6[6024] = {X 274.4972, Y 54.3961, Z -8.0000, A 0.000, B 0.000, C 0.000 }
gfCNCPoint6[6025] = {X 275.3426, Y 54.1003, Z -8.0000, A 0.000, B 0.000, C 0.000 }
gfCNCPoint6[6026] = {X 276.2327, Y 54.0000, Z -8.0000, A 0.000, B 0.000, C 0.000 }
gfCNCPoint6[6027] = {X 292.7731, Y 54.0000, Z -8.0000, A 0.000, B 0.000, C 0.000 }
gfCNCPoint6[6028] = {X 293.6632, Y 54.1003, Z -8.0000, A 0.000, B 0.000, C 0.000 }
gfCNCPoint6[6029] = {X 294.5086, Y 54.3961, Z -8.0000, A 0.000, B 0.000, C 0.000 }
gfCNCPoint6[6030] = {X 295.2670, Y 54.8727, Z -8.0000, A 0.000, B 0.000, C 0.000 }
gfCNCPoint6[6031] = {X 295.9004, Y 55.5060, Z -8.0000, A 0.000, B 0.000, C 0.000 }
gfCNCPoint6[6032] = {X 296.3770, Y 56.2645, Z -8.0000, A 0.000, B 0.000, C 0.000 }
gfCNCPoint6[6033] = {X 296.6728, Y 57.1099, Z -8.0000, A 0.000, B 0.000, C 0.000 }
gfCNCPoint6[6034] = {X 296.7731, Y 58.0000, Z -8.0000, A 0.000, B 0.000, C 0.000 }
gfCNCPoint6[6035] = {X 296.7731, Y 58.9341, Z -8.0000, A 0.000, B 0.000, C 0.000 }
gfCNCPoint6[6036] = {X 296.6603, Y 59.8687, Z -8.0000, A 0.000, B 0.000, C 0.000 }
gfCNCPoint6[6037] = {X 296.3330, Y 60.7513, Z -8.0000, A 0.000, B 0.000, C 0.000 }
gfCNCPoint6[6038] = {X 295.8093, Y 61.5335, Z -8.0000, A 0.000, B 0.000, C 0.000 }
gfCNCPoint6[6039] = {X 295.1178, Y 62.1723, Z -8.0000, A 0.000, B 0.000, C 0.000 }
gfCNCPoint6[6040] = {X 294.2967, Y 62.6326, Z -8.0000, A 0.000, B 0.000, C 0.000 }
gfCNCPoint6[6041] = {X 293.3910, Y 62.8891, Z -8.0000, A 0.000, B 0.000, C 0.000 }
gfCNCPoint6[6042] = {X 293.2334, Y 62.9110, Z -8.0000, A 0.000, B 0.000, C 0.000 }
gfCNCPoint6[6043] = {X 293.0752, Y 62.9268, Z -8.0000, A 0.000, B 0.000, C 0.000 }
gfCNCPoint6[6044] = {X 293.0541, Y 63.1540, Z -8.0000, A 0.000, B 0.000, C 0.000 }
gfCNCPoint6[6045] = {X 293.0541, Y 92.9237, Z -8.0000, A 0.000, B 0.000, C 0.000 }
gfCNCPoint6[6046] = {X 293.0752, Y 93.0658, Z -8.0000, A 0.000, B 0.000, C 0.000 }
gfCNCPoint6[6047] = {X 293.2328, Y 93.0820, Z -8.0000, A 0.000, B 0.000, C 0.000 }
gfCNCPoint6[6048] = {X 293.3897, Y 93.1045, Z -8.0000, A 0.000, B 0.000, C 0.000 }
gfCNCPoint6[6049] = {X 294.2952, Y 93.3636, Z -8.0000, A 0.000, B 0.000, C 0.000 }
gfCNCPoint6[6050] = {X 295.1159, Y 93.8256, Z -8.0000, A 0.000, B 0.000, C 0.000 }
gfCNCPoint6[6051] = {X 295.8071, Y 94.4655, Z -8.0000, A 0.000, B 0.000, C 0.000 }
gfCNCPoint6[6052] = {X 296.3309, Y 95.2482, Z -8.0000, A 0.000, B 0.000, C 0.000 }
gfCNCPoint6[6053] = {X 296.6589, Y 96.1311, Z -8.0000, A 0.000, B 0.000, C 0.000 }
gfCNCPoint6[6054] = {X 296.7731, Y 97.0660, Z -8.0000, A 0.000, B 0.000, C 0.000 }
gfCNCPoint6[6055] = {X 296.7731, Y 98.0000, Z -8.0000, A 0.000, B 0.000, C 0.000 }
gfCNCPoint6[6056] = {X 296.6728, Y 98.8901, Z -8.0000, A 0.000, B 0.000, C 0.000 }
gfCNCPoint6[6057] = {X 296.3770, Y 99.7355, Z -8.0000, A 0.000, B 0.000, C 0.000 }
gfCNCPoint6[6058] = {X 295.9004, Y 100.4940, Z -8.0000, A 0.000, B 0.000, C 0.000 }
gfCNCPoint6[6059] = {X 295.2670, Y 101.1273, Z -8.0000, A 0.000, B 0.000, C 0.000 }
gfCNCPoint6[6060] = {X 294.5086, Y 101.6039, Z -8.0000, A 0.000, B 0.000, C 0.000 }
gfCNCPoint6[6061] = {X 293.6632, Y 101.8997, Z -8.0000, A 0.000, B 0.000, C 0.000 }
gfCNCPoint6[6062] = {X 292.7731, Y 102.0000, Z -8.0000, A 0.000, B 0.000, C 0.000 }
gfCNCPoint6[6063] = {X 276.2327, Y 102.0000, Z -8.0000, A 0.000, B 0.000, C 0.000 }
gfCNCPoint6[6064] = {X 275.3426, Y 101.8997, Z -8.0000, A 0.000, B 0.000, C 0.000 }
